(* CODESYS project 轮毂电机.project

Project tree, tasks and I/O mapping:
  Device : AM521-0808TP/TN, Shenzhen Inovance Control Technology, version 3.5.11.50
      settings: PersistentStartAdddr = 0; PersistentStartEndAddr = 524287; Mode = 0
    application Application
      libraries: Standard, * (System); IoDrvCANopenAxis, 1.11.4.0 (Inovance); HC_CANBus, 0.1.3.0 (Inovance); Util, 3.5.11.0 (System); SM3_Drive_ETC_Inovance, 1.0.5.0 (Inovance)
      task MainTask (cyclic, interval t#4ms, priority 1) calls main
      task CANOPEN (cyclic, interval t#10ms, priority 2) calls CANOpen_Task
      program main [ST]
      DifferentialMonitor
      program CANOpen_Task [ST]
      global variables GVL
      function block FB_AckermannKinematics [ST]
      trace Trace (task MainTask): Rr_Wheel.diActVelocity
      function block FB_CommandLimiter [ST]
      function block FB_SteerPositionPID [ST]
      function block FB_RearWheelVelocityPID [ST]
      function block FB_AckermannInverseKinematics [ST]
      function block FB_UDP [ST]
      function block FB_PWM [ST]
      function block FB_CAN_SCU_1 [ST]
      function block FB_Test [ST]
      function block FB_MoveByYaokong [ST]
      function block FB_MoveByFSD [ST]
      function block FB_CAN_CCU [ST]
      function block FB_UDP_Recv [ST]
      function block FB_UDP_Send [ST]
      function block test [ST]
      function block FB_CAN_VCU_SES_Req [ST]
      function block FB_CAN_BMS [ST]
      function block cantesttest [LD]
    ConfigStorage
    Resources List
    Device Diagnosis
    Network Configuration
      LocalBus Config
    HardWare Configuration
    SoftMotion General Axis Pool
    Local Bus
      GL20_2CAN : GL20 2通道CAN通信接口模块, Inovance, order no. 01440308, version 00.00.00.10
          settings: ModuleBaseInfoStruct.BusType = 10; ModuleBaseInfoStruct.RackNumber = 1; ModuleBaseInfoStruct.SlotNumber = 1; COMPort1 = 32; COMPort2 = 33; devGuid1 = 'e5bf4089-cd92-4763-8943-9d7dacf300b6'; devGuid2 = '326b6049-3dfc-42ac-adce-35d035554d5f'
          unmapped channels: RxPDO_CH, TxPDO_CH
    CAN : CAN总线, INOVANCE, version 00.00.00.10
      CAN_Port : CAN Port, Inovance, version 00.00.00.10
          settings: IsFreeCAN = False; DeviceGuid = '83de0e76-e450-4053-a235-86c09473ce3d'; DeviceName = 'GE20_CAN_485'; InterfaceNo = 1; Device = 'AM521-0808TP/TN'; Port = 4; Type = 41108
        CANopen主站 : CANopen主站, Inovance, version 00.00.00.10
            settings: COPManagerSyncStruct.SyncType = 1; COPManagerSyncStruct.SyncPeriod = 10000; COPManagerHeartbeatStruct.Enable = 1; Port NO = 4; IsPortSub = True; IsMainCAN = False; IsCANExt = True; IsLocalCAN = False
          C6049 : CANopen Slaver, Inovance, order no. 1525, version 00.00.00.10
              settings: NodeID = 3; EnableExpertSettings = 1; Error Control.SlaveHeartbeat.ProduceTime = 300; Error Control.SlaveHeartbeat.NrofConsumer = 1; VendorID = 1097; ProductNumber = 1; RevisionNumber = 131075; NrofRxPDO = 4; ValidRxPDO = 2; PdoCommuIndex = 5120; CanId = 515; TxType = 255;  = 1;  = 805306432; PdoCommuIndex = 5121; CanId = 771; TxType = 255;  = 1;  = 805371968; PdoCommuIndex = 5122; CanId = 1027; TxType = 255;  = 1;  = 805437504; PdoCommuIndex = 5123; CanId = 1283; TxType = 255;  = 1;  = 805503040; NrofTxPDO = 4; ValidTxPDO = 3; PdoCommuIndex = 6144; CanId = 387; TxType = 255; InhibitTime = 50;  = 1;  = 805568576; PdoCommuIndex = 6145; CanId = 643; TxType = 255;
                InhibitTime = 50;  = 1;  = 805634112; PdoCommuIndex = 6146; CanId = 899; TxType = 255; InhibitTime = 50;  = 1;  = 805699648; PdoCommuIndex = 6147; CanId = 1155; TxType = 255; InhibitTime = 50;  = 1;  = 805765184; SdoTimeout = 1000; NrofSDO = 31; SdoCommParam = 269877536; SdoErrHandle = 2; SdoJumptoLine = 31; SdoCommParam = 269942800; SdoCommValue = 300; SdoErrHandle = 2; SdoJumptoLine = 31; SdoCommParam = 269746208; SdoCommValue = 2147483779; SdoErrHandle = 2; SdoJumptoLine = 31; SdoCommParam = 269746208; SdoCommValue = 131; SdoErrHandle = 2; SdoJumptoLine = 31; SdoCommParam = 335544608; SdoCommValue = 2147484163; SdoErrHandle = 2; SdoJumptoLine = 31; SdoCommParam = 335610144; SdoCommValue = 2147484419; SdoErrHandle = 2; SdoJumptoLine = 31;
                SdoCommParam = 335610376; SdoCommValue = 255; SdoErrHandle = 2; SdoJumptoLine = 31; SdoCommParam = 369164296; SdoErrHandle = 2; SdoJumptoLine = 31; SdoCommParam = 369164576; SdoCommValue = 805371968; SdoErrHandle = 2; SdoJumptoLine = 31; SdoCommParam = 369164296; SdoCommValue = 1; SdoErrHandle = 2; SdoJumptoLine = 31; SdoCommParam = 335610144; SdoCommValue = 771; SdoErrHandle = 2; SdoJumptoLine = 31; SdoCommParam = 335675680; SdoCommValue = 2147484675; SdoErrHandle = 2; SdoJumptoLine = 31; SdoCommParam = 335741216; SdoCommValue = 2147484931; SdoErrHandle = 2; SdoJumptoLine = 31; SdoCommParam = 402653472; SdoCommValue = 2147484035; SdoErrHandle = 2; SdoJumptoLine = 31; SdoCommParam = 402653704; SdoCommValue = 255; SdoErrHandle = 2; SdoJumptoLine = 31; SdoCommParam = 402653968; SdoCommValue = 50; SdoErrHandle = 2; SdoJumptoLine = 31; SdoCommParam = 402654480;
                SdoErrHandle = 2; SdoJumptoLine = 31; SdoCommParam = 436207624; SdoErrHandle = 2; SdoJumptoLine = 31; SdoCommParam = 436207904; SdoCommValue = 805568576; SdoErrHandle = 2; SdoJumptoLine = 31; SdoCommParam = 436207624; SdoCommValue = 1; SdoErrHandle = 2; SdoJumptoLine = 31; SdoCommParam = 402653472; SdoCommValue = 387; SdoErrHandle = 2; SdoJumptoLine = 31; SdoCommParam = 402719008; SdoCommValue = 2147484291; SdoErrHandle = 2; SdoJumptoLine = 31; SdoCommParam = 402719240; SdoCommValue = 255; SdoErrHandle = 2; SdoJumptoLine = 31; SdoCommParam = 402719504; SdoCommValue = 50; SdoErrHandle = 2; SdoJumptoLine = 31; SdoCommParam = 402720016; SdoErrHandle = 2; SdoJumptoLine = 31; SdoCommParam = 436273160; SdoErrHandle = 2; SdoJumptoLine = 31; SdoCommParam = 436273440; SdoCommValue = 805634112; SdoErrHandle = 2; SdoJumptoLine = 31; SdoCommParam = 436273160;
                SdoCommValue = 1; SdoErrHandle = 2; SdoJumptoLine = 31; SdoCommParam = 402719008; SdoCommValue = 643; SdoErrHandle = 2; SdoJumptoLine = 31; SdoCommParam = 402784544; SdoCommValue = 2147484547; SdoErrHandle = 2; SdoJumptoLine = 31; SdoCommParam = 402850080; SdoCommValue = 2147484803; SdoErrHandle = 2; SdoJumptoLine = 31; FileName = 'C6049.eds'; FileVersion = '0x02'; FileRevision = '0x01'; EDSVersion = '4.0'; Description = 'EDS for 6049  Canopen Slave'; EDS File Path = 'D:\Asoftware\InoProShop\CODESYS\Common\AM600 Data\EdsFile\C6049.eds'; EDSVersion = 'EDLS'; VendorNumber = 1097; ProductName = 'C6049'; ProductNumber = 1; RevisionNumber = 131075; OrderCode = '60'; Baudrate = 368; SimpleBootUpSlave = 1; Granularity = 0; DynamicChannelsSupported = 0; GroupMessaging = 0; NrOfRXPDO = 4; NrOfTXPDO = 4; LSS_Supported = 0; DummyUsage = 0; SDOType = 0; SDOName = 'Set Heartbeat Consumer'; SDOType = 0; SDOName = 'Set Heartbeat Producer';
                SDOType = 0; SDOName = 'Disable Emcy COB-ID'; SDOType = 0; SDOName = 'Set Emcy COB-ID'; SDOType = 0; SDOName = 'Disable PDO'; SDOType = 0; SDOName = 'Disable PDO'; SDOType = 0; SDOName = 'Set transmission type'; SDOType = 0; SDOName = 'Clear PDO mapping'; SDOType = 0; SDOName = 'Set mapping'; SDOType = 0; SDOName = 'Set number of pdos'; SDOType = 0; SDOName = 'Set and enable COB-ID'; SDOType = 0; SDOName = 'Disable PDO'; SDOType = 0; SDOName = 'Disable PDO'; SDOType = 0; SDOName = 'Disable PDO'; SDOType = 0; SDOName = 'Set transmission type'; SDOType = 0; SDOName = 'Set inhibit time'; SDOType = 0; SDOName = 'Set event time'; SDOType = 0; SDOName = 'Clear PDO mapping'; SDOType = 0; SDOName = 'Set mapping'; SDOType = 0; SDOName = 'Set number of pdos'; SDOType = 0; SDOName = 'Set and enable COB-ID'; SDOType = 0; SDOName = 'Disable PDO';
                SDOType = 0; SDOName = 'Set transmission type'; SDOType = 0; SDOName = 'Set inhibit time'; SDOType = 0; SDOName = 'Set event time'; SDOType = 0; SDOName = 'Clear PDO mapping'; SDOType = 0; SDOName = 'Set mapping'; SDOType = 0; SDOName = 'Set number of pdos'; SDOType = 0; SDOName = 'Set and enable COB-ID'; SDOType = 0; SDOName = 'Disable PDO'; SDOType = 0; SDOName = 'Disable PDO'; Recv PDO Mapping Name.Recv PDO Mapping Name = '64 DI0'; Recv PDO Mapping Name.Recv PDO Mapping Name = '64 DI1'; Recv PDO Mapping Name.Recv PDO Mapping Name = '64 AI0'; Recv PDO Mapping Name.Recv PDO Mapping Name = '64 AI1'; Send PDO Mapping Name.Send PDO Mapping Name = '64 DO0'; Send PDO Mapping Name.Send PDO Mapping Name = '64 DO1'; Send PDO Mapping Name.Send PDO Mapping Name = '64 AO0'; Send PDO Mapping Name.Send PDO Mapping Name = '64 AO1'; Is Manual change COB-ID = 0; Is Manual change COB-ID = 0; Is Manual change COB-ID = 0; Is Manual change COB-ID = 0; Is Manual change COB-ID = 0; Is Manual change COB-ID = 0; Is Manual change COB-ID = 0; Is Manual change COB-ID = 0; MandatoryObjs = 3; Object Dictionary Item = '1000;Device Type;0x00000000;7;7;RO;0;-1;-1;-1'; Object Dictionary Item = '1001;Error Register;0x0;5;7;RO;0;-1;-1;-1'; Object Dictionary Item = '1018;Identity Object;;-1;9;;-1;4;-1;-1'; Object Dictionary Item = '1018sub0;number of entries;3;5;7;RO;0;-1;4;1'; Object Dictionary Item = '1018sub1;Vendor ID;0x00000449;7;7;RO;0;-1;-1;-1';
                Object Dictionary Item = '1018sub2;Product code;0x00000001;7;7;RO;0;-1;-1;-1'; Object Dictionary Item = '1018sub3;Revision number;0x00020003;7;7;RO;0;-1;-1;-1'; ManufacturerObjs = 9; Object Dictionary Item = '2000;Index 0x2000;;-1;9;;-1;2;-1;-1'; Object Dictionary Item = '2000sub0;Set TXPDO inhibit time;0x01;5;7;RO;0;-1;-1;-1'; Object Dictionary Item = '2000sub1;TXPDO1 inhibit time;100;5;7;RW;0;-1;-1;-1'; Object Dictionary Item = '3000;64 DI0;0;27;7;RO;1;-1;-1;-1'; Object Dictionary Item = '3001;64 DI1;0x0;27;7;RO;1;-1;-1;-1'; Object Dictionary Item = '3002;64 AI0;0;27;7;RO;1;-1;-1;-1'; Object Dictionary Item = '3003;64 AI1;0x0;27;7;RO;1;-1;-1;-1'; Object Dictionary Item = '3004;64 DO0;0x0;27;7;RWW;1;-1;-1;-1'; Object Dictionary Item = '3005;64 DO1;0x0;27;7;RWW;1;-1;-1;-1'; Object Dictionary Item = '3006;64 AO0;0x0;27;7;RWW;1;-1;-1;-1'; Object Dictionary Item = '3007;64 AO1;0x0;27;7;RWW;1;-1;-1;-1'; OptionsObjs = 20; Object Dictionary Item = '1005;COB-ID SYNC message;0x80;7;7;RW;0;-1;-1;-1'; Object Dictionary Item = '1008;Device Name;4055;9;7;CONST;0;-1;-1;-1'; Object Dictionary Item = '1016;Consumer Heartbeat time group;;-1;8;;-1;2;-1;-1'; Object Dictionary Item = '1016sub0;Number of entries;1;5;7;RO;0;-1;-1;-1'; Object Dictionary Item = '1016sub1;Consumer Heartbeat time;0;7;7;RW;0;-1;-1;-1'; Object Dictionary Item = '1017;Producer Heartbeat time group;0;6;7;RW;0;-1;-1;-1'; Object Dictionary Item = '1400;Receive PDO1 parameter;;-1;9;;-1;4;-1;-1'; Object Dictionary Item = '1400sub0;Number of entries;3;5;7;RO;0;-1;-1;-1'; Object Dictionary Item = '1400sub1;COB-ID;$NodeID + 0x200;7;7;RW;0;-1;-1;-1'; Object Dictionary Item = '1400sub2;Transmission type;255;5;7;RW;0;-1;-1;-1'; Object Dictionary Item = '1400sub3;Inhibit timer;0;5;7;RW;0;-1;-1;-1'; Object Dictionary Item = '1600;Receive PDO1 mapping;;-1;9;;-1;2;-1;-1'; Object Dictionary Item = '1600sub0;Number of mapped objects;0x1;5;7;RO;0;-1;5;0'; Object Dictionary Item = '1600sub1;1.mapped object;0x30000040;7;7;RO;0;-1;-1;-1'; Object Dictionary Item = '1401;Receive PDO2 parameter;;-1;9;;-1;4;-1;-1'; Object Dictionary Item = '1401sub0;Number of entries;3;5;7;RO;0;-1;-1;-1'; Object Dictionary Item = '1401sub1;COB-ID;$NodeID + 0x300;7;7;RW;0;-1;-1;-1'; Object Dictionary Item = '1401sub2;Transmission type;255;5;7;RW;0;-1;-1;-1'; Object Dictionary Item = '1401sub3;Inhibit timer;0;5;7;RW;0;-1;-1;-1'; Object Dictionary Item = '1601;Receive PDO2 mapping;;-1;9;;-1;2;-1;-1'; Object Dictionary Item = '1601sub0;Number of mapped objects;0x1;5;7;RO;0;-1;5;0'; Object Dictionary Item = '1601sub1;1.mapped object;0x30010040;7;7;RO;0;-1;-1;-1'; Object Dictionary Item = '1402;Receive PDO3 parameter;;-1;9;;-1;4;-1;-1'; Object Dictionary Item = '1402sub0;Number of entries;3;5;7;RO;0;-1;-1;-1'; Object Dictionary Item = '1402sub1;COB-ID;$NodeID + 0x400;7;7;RW;0;-1;-1;-1';
                Object Dictionary Item = '1402sub2;Transmission type;255;5;7;RW;0;-1;-1;-1'; Object Dictionary Item = '1402sub3;Inhibit timer;0;5;7;RW;0;-1;-1;-1'; Object Dictionary Item = '1602;Receive PDO3 mapping;;-1;9;;-1;2;-1;-1'; Object Dictionary Item = '1602sub0;Number of mapped objects;0x1;5;7;RO;0;-1;5;0'; Object Dictionary Item = '1602sub1;1.mapped object;0x30020040;7;7;RO;0;-1;-1;-1'; Object Dictionary Item = '1403;Receive PDO4 parameter;;-1;9;;-1;4;-1;-1'; Object Dictionary Item = '1403sub0;Number of entries;3;5;7;RO;0;-1;-1;-1'; Object Dictionary Item = '1403sub1;COB-ID;$NodeID + 0x500;7;7;RW;0;-1;-1;-1'; Object Dictionary Item = '1403sub2;Transmission type;255;5;7;RW;0;-1;-1;-1'; Object Dictionary Item = '1403sub3;Inhibit timer;0;5;7;RW;0;-1;-1;-1'; Object Dictionary Item = '1603;Receive PDO4 mapping;;-1;9;;-1;2;-1;-1'; Object Dictionary Item = '1603sub0;Number of mapped objects;0x1;5;7;RO;0;-1;5;0'; Object Dictionary Item = '1603sub1;1.mapped object;0x30030040;7;7;RO;0;-1;-1;-1'; Object Dictionary Item = '1800;Transmit PDO1 parameter;;-1;9;;-1;5;-1;-1'; Object Dictionary Item = '1800sub0;Number of entries;0x5;5;7;RO;0;-1;-1;-1'; Object Dictionary Item = '1800sub1;COB-ID;$NodeID + 0x180;7;7;RW;0;-1;-1;-1'; Object Dictionary Item = '1800sub2;Transmission type;255;5;7;RW;0;-1;-1;-1'; Object Dictionary Item = '1800sub3;Inhibit timer;50;6;7;RW;0;-1;-1;-1'; Object Dictionary Item = '1800sub5;Event Timer;0;27;7;RW;0;-1;65535;0'; Object Dictionary Item = '1A00;Transmit PDO1 mapping;;-1;9;;-1;2;-1;-1'; Object Dictionary Item = '1A00sub0;Number of mapped objects;0x1;5;7;RO;0;-1;4;0'; Object Dictionary Item = '1A00sub1;1.mapped object;0x30040040;7;7;RO;0;-1;-1;-1'; Object Dictionary Item = '1801;Transmit PDO2 parameter;;-1;9;;-1;5;-1;-1'; Object Dictionary Item = '1801sub0;Number of entries;0x5;5;7;RO;0;-1;-1;-1'; Object Dictionary Item = '1801sub1;COB-ID;$NodeID + 0x280;7;7;RW;0;-1;-1;-1'; Object Dictionary Item = '1801sub2;Transmission type;255;5;7;RW;0;-1;-1;-1'; Object Dictionary Item = '1801sub3;Inhibit timer;50;6;7;RW;0;-1;-1;-1'; Object Dictionary Item = '1801sub5;Event Timer;0;27;7;RW;0;-1;65535;0'; Object Dictionary Item = '1A01;Transmit PDO2 mapping;;-1;9;;-1;2;-1;-1'; Object Dictionary Item = '1A01sub0;Number of mapped objects;0x1;5;7;RO;0;-1;4;0'; Object Dictionary Item = '1A01sub1;1.mapped object;0x30050040;7;7;RO;0;-1;-1;-1'; Object Dictionary Item = '1802;Transmit PDO3 parameter;;-1;9;;-1;5;-1;-1'; Object Dictionary Item = '1802sub0;Number of entries;0x5;5;7;RO;0;-1;-1;-1'; Object Dictionary Item = '1802sub1;COB-ID;$NodeID + 0x380;7;7;RW;0;-1;-1;-1'; Object Dictionary Item = '1802sub2;Transmission type;255;5;7;RW;0;-1;-1;-1'; Object Dictionary Item = '1802sub3;Inhibit timer;50;6;7;RW;0;-1;-1;-1'; Object Dictionary Item = '1802sub5;Event Timer;0;27;7;RW;0;-1;65535;0'; Object Dictionary Item = '1A02;Transmit PDO3 mapping;;-1;9;;-1;2;-1;-1'; Object Dictionary Item = '1A02sub0;Number of mapped objects;0x1;5;7;RO;0;-1;4;0'; Object Dictionary Item = '1A02sub1;1.mapped object;0x30060040;7;7;RO;0;-1;-1;-1';
                Object Dictionary Item = '1803;Transmit PDO4 parameter;;-1;9;;-1;5;-1;-1'; Object Dictionary Item = '1803sub0;Number of entries;0x5;5;7;RO;0;-1;-1;-1'; Object Dictionary Item = '1803sub1;COB-ID;$NodeID + 0x480;7;7;RW;0;-1;-1;-1'; Object Dictionary Item = '1803sub2;Transmission type;255;5;7;RW;0;-1;-1;-1'; Object Dictionary Item = '1803sub3;Inhibit timer;50;6;7;RW;0;-1;-1;-1'; Object Dictionary Item = '1803sub5;Event Timer;0;27;7;RW;0;-1;65535;0'; Object Dictionary Item = '1A03;Transmit PDO4 mapping;;-1;9;;-1;2;-1;-1'; Object Dictionary Item = '1A03sub0;Number of mapped objects;0x1;5;7;RO;0;-1;4;0'; Object Dictionary Item = '1A03sub1;1.mapped object;0x30070040;7;7;RO;0;-1;-1;-1'
              output Application.YkqRxPDO0_data : LWORD  // 64 DI1
              input  Application.YkqTxPDO0_data : LWORD  // 64 DO0
              input  Application.Emergency_Stop : BOOL  // 64 DO0.Bit0
              input  Application.DriveByYaokong : BOOL  // 64 DO0.Bit10
              input  Application.DriveBySelf : BOOL  // 64 DO0.Bit11
              input  Application.Remote_Break : BOOL  // 64 DO0.Bit15
              input  Application.YkqTxPDO1_data : LWORD  // 64 DO1
          FDKServo_PMSM : CANopen Slaver, Inovance, order no. 1525, version 00.00.00.10
              settings: NodeID = 2; EnableExpertSettings = 1; Error Control.SlaveHeartbeat.ProduceTime = 300; Error Control.SlaveHeartbeat.NrofConsumer = 1; DeviceType = 131474; VendorID = 1459275; ProductNumber = 66128; NrofRxPDO = 4; ValidRxPDO = 3; PdoCommuIndex = 5120; CanId = 514; TxType = 255;  = 3;  = 1614807056;  = 1627324448;  = 1616904200; PdoCommuIndex = 5121; CanId = 770; TxType = 255;  = 2;  = 1618608160;  = 1619001376; PdoCommuIndex = 5122; CanId = 1026; TxType = 255;  = 0; PdoCommuIndex = 5123; CanId = 1282; TxType = 255;  = 0; NrofTxPDO = 4; ValidTxPDO = 3; PdoCommuIndex = 6144; CanId = 386; TxType = 255; InhibitTime = 100; EventTime = 10;  = 4;  = 1614872592;  = 536870928;
                 = 536936464;  = 1616969736; PdoCommuIndex = 6145; CanId = 642; TxType = 255; InhibitTime = 100; EventTime = 10;  = 2;  = 1617166368;  = 1617690656; PdoCommuIndex = 6146; CanId = 898; TxType = 255; InhibitTime = 100; EventTime = 10;  = 0; PdoCommuIndex = 6147; CanId = 1154; TxType = 255; InhibitTime = 100; EventTime = 10;  = 0; SdoTimeout = 1000; NrofSDO = 44; SdoCommParam = 268763168; SdoCommValue = 128; SdoCommParam = 269877536; SdoCommParam = 269942800; SdoCommValue = 300; SdoCommParam = 269746208; SdoCommValue = 2147483778; SdoCommParam = 269746208; SdoCommValue = 130; SdoCommParam = 335544608; SdoCommValue = 2147484162; SdoCommParam = 335544840; SdoCommValue = 255; SdoCommParam = 369098760; SdoCommParam = 369099040; SdoCommValue = 1614807056;
                SdoCommParam = 369099296; SdoCommValue = 1627324448; SdoCommParam = 369099552; SdoCommValue = 1616904200; SdoCommParam = 369098760; SdoCommValue = 3; SdoCommParam = 335544608; SdoCommValue = 514; SdoCommParam = 335610144; SdoCommValue = 2147484418; SdoCommParam = 335610376; SdoCommValue = 255; SdoCommParam = 369164296; SdoCommParam = 369164576; SdoCommValue = 1618608160; SdoCommParam = 369164832; SdoCommValue = 1619001376; SdoCommParam = 369164296; SdoCommValue = 2; SdoCommParam = 335610144; SdoCommValue = 770; SdoCommParam = 335675680; SdoCommValue = 2147484674; SdoCommParam = 335741216; SdoCommValue = 2147484930; SdoCommParam = 402653472; SdoCommValue = 2147484034; SdoCommParam = 402653704; SdoCommValue = 255; SdoCommParam = 402653968; SdoCommValue = 100; SdoCommParam = 402654480; SdoCommValue = 10; SdoCommParam = 436207624; SdoCommParam = 436207904; SdoCommValue = 1614872592; SdoCommParam = 436208160; SdoCommValue = 536870928; SdoCommParam = 436208416; SdoCommValue = 536936464;
                SdoCommParam = 436208672; SdoCommValue = 1616969736; SdoCommParam = 436207624; SdoCommValue = 4; SdoCommParam = 402653472; SdoCommValue = 386; SdoCommParam = 402719008; SdoCommValue = 2147484290; SdoCommParam = 402719240; SdoCommValue = 255; SdoCommParam = 402719504; SdoCommValue = 100; SdoCommParam = 402720016; SdoCommValue = 10; SdoCommParam = 436273160; SdoCommParam = 436273440; SdoCommValue = 1617166368; SdoCommParam = 436273696; SdoCommValue = 1617690656; SdoCommParam = 436273160; SdoCommValue = 2; SdoCommParam = 402719008; SdoCommValue = 642; SdoCommParam = 402784544; SdoCommValue = 2147484546; SdoCommParam = 402850080; SdoCommValue = 2147484802; FileName = 'FDK_PMSM.eds'; FileVersion = '0x01'; FileRevision = '0x01'; EDSVersion = '4.0'; Description = 'EDS for FDK_Single_DRIVER'; EDS File Path = 'D:\Asoftware\InoProShop\CODESYS\Common\AM600 Data\EdsFile\FDK_PMSM_SIEMENS-VSXXDXX-A-20240203.eds'; EDSVersion = 'FDK, INC.'; VendorNumber = 1459275; ProductName = 'FDKServo-PMSM'; ProductNumber = 66128; RevisionNumber = 0; OrderCode = 'DVPCOPM-SL'; Baudrate = 503;
                SimpleBootUpSlave = 1; Granularity = 8; DynamicChannelsSupported = 0; GroupMessaging = 0; NrOfRXPDO = 4; NrOfTXPDO = 4; LSS_Supported = 1; DummyUsage = 0; SDOType = 0; SDOName = 'Disable COB-ID sync'; SDOType = 0; SDOName = 'Set Heartbeat Consumer'; SDOType = 0; SDOName = 'Set Heartbeat Producer'; SDOType = 0; SDOName = 'Disable Emcy COB-ID'; SDOType = 0; SDOName = 'Set Emcy COB-ID'; SDOType = 0; SDOName = 'Disable PDO'; SDOType = 0; SDOName = 'Set transmission type'; SDOType = 0; SDOName = 'Clear PDO mapping'; SDOType = 0; SDOName = 'Set mapping'; SDOType = 0; SDOName = 'Set mapping'; SDOType = 0; SDOName = 'Set mapping'; SDOType = 0; SDOName = 'Set number of pdos'; SDOType = 0; SDOName = 'Set and enable COB-ID'; SDOType = 0; SDOName = 'Disable PDO'; SDOType = 0; SDOName = 'Set transmission type'; SDOType = 0; SDOName = 'Clear PDO mapping';
                SDOType = 0; SDOName = 'Set mapping'; SDOType = 0; SDOName = 'Set mapping'; SDOType = 0; SDOName = 'Set number of pdos'; SDOType = 0; SDOName = 'Set and enable COB-ID'; SDOType = 0; SDOName = 'Disable PDO'; SDOType = 0; SDOName = 'Disable PDO'; SDOType = 0; SDOName = 'Disable PDO'; SDOType = 0; SDOName = 'Set transmission type'; SDOType = 0; SDOName = 'Set inhibit time'; SDOType = 0; SDOName = 'Set event time'; SDOType = 0; SDOName = 'Clear PDO mapping'; SDOType = 0; SDOName = 'Set mapping'; SDOType = 0; SDOName = 'Set mapping'; SDOType = 0; SDOName = 'Set mapping'; SDOType = 0; SDOName = 'Set mapping'; SDOType = 0; SDOName = 'Set number of pdos'; SDOType = 0; SDOName = 'Set and enable COB-ID'; SDOType = 0; SDOName = 'Disable PDO'; SDOType = 0; SDOName = 'Set transmission type'; SDOType = 0; SDOName = 'Set inhibit time';
                SDOType = 0; SDOName = 'Set event time'; SDOType = 0; SDOName = 'Clear PDO mapping'; SDOType = 0; SDOName = 'Set mapping'; SDOType = 0; SDOName = 'Set mapping'; SDOType = 0; SDOName = 'Set number of pdos'; SDOType = 0; SDOName = 'Set and enable COB-ID'; SDOType = 0; SDOName = 'Disable PDO'; SDOType = 0; SDOName = 'Disable PDO'; Recv PDO Mapping Name.Recv PDO Mapping Name = 'Controlword'; Recv PDO Mapping Name.Recv PDO Mapping Name = 'Target Velocity'; Recv PDO Mapping Name.Recv PDO Mapping Name = 'Modes of operation'; Recv PDO Mapping Name.Recv PDO Mapping Name = 'Target Position'; Recv PDO Mapping Name.Recv PDO Mapping Name = 'Max motor speed'; Send PDO Mapping Name.Send PDO Mapping Name = 'Statusword'; Send PDO Mapping Name.Send PDO Mapping Name = 'FaultCode1'; Send PDO Mapping Name.Send PDO Mapping Name = 'WorkState1'; Send PDO Mapping Name.Send PDO Mapping Name = 'Modes Of Operation Display'; Send PDO Mapping Name.Send PDO Mapping Name = 'Position Actual Value'; Send PDO Mapping Name.Send PDO Mapping Name = 'Velocity actual value'; Is Manual change COB-ID = 0; Is Manual change COB-ID = 0; Is Manual change COB-ID = 0; Is Manual change COB-ID = 0; Is Manual change COB-ID = 0; Is Manual change COB-ID = 0; Is Manual change COB-ID = 0; Is Manual change COB-ID = 0; MandatoryObjs = 3; Object Dictionary Item = '1000;CAN Controller Type;0x20192;7;7;RO;0;-1;-1;-1'; Object Dictionary Item = '1001;Error Register;0;5;7;RO;0;-1;-1;-1'; Object Dictionary Item = '1018;Identity Object;;-1;9;;-1;4;-1;-1'; Object Dictionary Item = '1018sub0;number of entries;3;5;7;RO;0;-1;4;1';
                Object Dictionary Item = '1018sub1;Vendor ID;0x0016444B;7;7;RO;0;-1;-1;-1'; Object Dictionary Item = '1018sub2;Product code;0x00010250;7;7;RO;0;-1;-1;-1'; Object Dictionary Item = '1018sub3;Revision number;0x00000000;7;7;RO;0;-1;-1;-1'; ManufacturerObjs = 30; Object Dictionary Item = '2000;FaultCode1;;6;7;RO;1;-1;65535;0'; Object Dictionary Item = '2001;WorkState1;;6;7;RO;1;-1;65535;0'; Object Dictionary Item = '2002;Motor_T;;6;7;RO;1;-1;-1;-1'; Object Dictionary Item = '2004;WARN;;6;7;RO;1;-1;65535;0'; Object Dictionary Item = '2005;CurrentBase;;6;7;RO;1;-1;65535;0'; Object Dictionary Item = '2006;LineEncoder;;4;7;RO;1;-1;65535;0'; Object Dictionary Item = '2007;Feedback Type;;6;7;RW;0;-1;65535;0'; Object Dictionary Item = '2008;Pole Pairs;;6;7;RW;0;-1;65535;0'; Object Dictionary Item = '2009;CAN ID;;5;7;RW;0;-1;-1;-1'; Object Dictionary Item = '200A;Can Baud Rate;;6;7;RW;0;-1;-1;-1'; Object Dictionary Item = '200B;Rated Current;;3;7;RW;0;-1;-1;-1'; Object Dictionary Item = '200C;Rated Speed;;3;7;RW;0;-1;-1;-1'; Object Dictionary Item = '200D;Overload Current;;6;7;RW;1;-1;-1;-1'; Object Dictionary Item = '200E;Overload Time;;6;7;RW;1;-1;-1;-1'; Object Dictionary Item = '200F;Current Loop P;;6;7;RW;1;-1;-1;-1'; Object Dictionary Item = '2010;Current Loop I;;6;7;RW;1;-1;-1;-1'; Object Dictionary Item = '2011;Speed Loop p0;;6;7;RW;1;-1;-1;-1'; Object Dictionary Item = '2012;Speed Loop P1;;6;7;RW;1;-1;-1;-1'; Object Dictionary Item = '2013;Speed Loop I;;6;7;RW;1;-1;-1;-1'; Object Dictionary Item = '2014;Position Loop P0;;6;7;RW;1;-1;-1;-1'; Object Dictionary Item = '2015;Position Loop P1;;6;7;RW;1;-1;-1;-1'; Object Dictionary Item = '2016;Command0;;6;7;RW;1;-1;-1;-1'; Object Dictionary Item = '2017;Command1;;6;7;RW;1;-1;-1;-1'; Object Dictionary Item = '2018;Software Limited Cache;;6;7;RW;1;-1;-1;-1'; Object Dictionary Item = '2019;Software Limited Forward Position;;4;7;RW;1;-1;-1;-1'; Object Dictionary Item = '201A;Software Limited Reverse Position;;4;7;RW;1;-1;-1;-1'; Object Dictionary Item = '201B;RS485_NodeID;;6;7;RW;1;-1;-1;-1'; Object Dictionary Item = '201C;RS485_Baudrate;;6;7;RW;1;-1;-1;-1'; Object Dictionary Item = '201D;RS485_Protocol;;6;7;RW;1;-1;-1;-1'; Object Dictionary Item = '22A2;System_T;;6;7;RO;1;-1;-1;-1'; OptionsObjs = 104; Object Dictionary Item = '1002;Manufacturer Status Register;;7;7;RO;1;-1;-1;-1'; Object Dictionary Item = '1003;Pre-defined Error Field;;-1;8;;-1;17;-1;-1'; Object Dictionary Item = '1003sub0;Number of Errors;0;5;7;RW;0;-1;16;0'; Object Dictionary Item = '1003sub1;Standard Error Field;0;7;7;RO;0;-1;-1;0'; Object Dictionary Item = '1003sub2;Standard Error Field;0;7;7;RO;0;-1;-1;0';
                Object Dictionary Item = '1003sub3;Standard Error Field;0;7;7;RO;0;-1;-1;0'; Object Dictionary Item = '1003sub4;Standard Error Field;0;7;7;RO;0;-1;-1;0'; Object Dictionary Item = '1003sub5;Standard Error Field;0;7;7;RO;0;-1;-1;0'; Object Dictionary Item = '1003sub6;Standard Error Field;0;7;7;RO;0;-1;-1;0'; Object Dictionary Item = '1003sub7;Standard Error Field;0;7;7;RO;0;-1;-1;0'; Object Dictionary Item = '1003sub8;Standard Error Field;0;7;7;RO;0;-1;-1;0'; Object Dictionary Item = '1003sub9;Standard Error Field;0;7;7;RO;0;-1;-1;0'; Object Dictionary Item = '1003suba;Standard Error Field;0;7;7;RO;0;-1;-1;0'; Object Dictionary Item = '1003subb;Standard Error Field;0;7;7;RO;0;-1;-1;0'; Object Dictionary Item = '1003subc;Standard Error Field;0;7;7;RO;0;-1;-1;0'; Object Dictionary Item = '1003subd;Standard Error Field;0;7;7;RO;0;-1;-1;0'; Object Dictionary Item = '1003sube;Standard Error Field;0;7;7;RO;0;-1;-1;0'; Object Dictionary Item = '1003subf;Standard Error Field;0;7;7;RO;0;-1;-1;0'; Object Dictionary Item = '1003sub10;Standard Error Field;0;7;7;RO;0;-1;-1;0'; Object Dictionary Item = '1005;COB-ID SYNC-message;0x80;7;7;RW;0;-1;-1;-1'; Object Dictionary Item = '1006;Communication Cycle Period;0;7;7;RW;0;-1;-1;0'; Object Dictionary Item = '1008;Manufacturer Device Name;;9;7;CONST;0;-1;-1;-1'; Object Dictionary Item = '1009;Manufacturer Hardware Version;;9;7;CONST;0;-1;-1;-1'; Object Dictionary Item = '100A;Manufacturer Software Version;;9;7;CONST;0;-1;-1;-1'; Object Dictionary Item = '100B;Node-ID;1;5;7;RO;0;-1;127;1'; Object Dictionary Item = '1010;Store Parameters;;-1;8;;-1;4;-1;-1'; Object Dictionary Item = '1010sub0;Largest Supported Sub-index;3;5;7;RO;0;-1;3;3'; Object Dictionary Item = '1010sub1;Save All Parameters;;7;7;RW;0;-1;-1;-1'; Object Dictionary Item = '1010sub2;Save Communication Parameters;0;7;7;RW;0;-1;-1;-1'; Object Dictionary Item = '1010sub3;Save ApplicationParameters;0;7;7;RW;0;-1;-1;-1'; Object Dictionary Item = '1011;Restore  Parameters;;-1;8;;-1;4;-1;-1'; Object Dictionary Item = '1011sub0;Largest Supported Sub-index;3;5;7;RO;0;-1;3;3'; Object Dictionary Item = '1011sub1;Restore All Parameters;;7;7;RW;0;-1;-1;-1'; Object Dictionary Item = '1011sub2;Restore Communication Parameters;0;7;7;RW;0;-1;-1;-1'; Object Dictionary Item = '1011sub3;Restore ApplicationParameters;0;7;7;RW;0;-1;-1;-1'; Object Dictionary Item = '1012;COB-ID Time Stamp Message;0x80000100;7;7;RW;0;-1;-1;-1'; Object Dictionary Item = '1013;High Resolution TimeStamp;0;7;7;RW;0;-1;-1;0'; Object Dictionary Item = '1014;COB-ID Emergency Message;$NODEID+0x80;7;7;RW;0;-1;-1;-1'; Object Dictionary Item = '1016;Consumer Heartbeat Time;;-1;8;;-1;2;-1;-1'; Object Dictionary Item = '1016sub0;Number of Entries;1;5;7;RO;0;-1;1;1'; Object Dictionary Item = '1016sub1;Consumer Heartbeat Time;0;7;7;RW;0;-1;-1;-1'; Object Dictionary Item = '1017;Producer heartbeat time;0;6;7;RW;0;-1;-1;-1'; Object Dictionary Item = '1023;OS Command;;-1;9;;-1;4;-1;-1'; Object Dictionary Item = '1023sub0;Number of Entries;3;5;7;RO;0;-1;3;3'; Object Dictionary Item = '1023sub1;Command;;10;7;WO;0;-1;-1;-1';
                Object Dictionary Item = '1023sub2;Status;0;5;7;RO;0;-1;255;0'; Object Dictionary Item = '1023sub3;Reply;;10;7;RO;0;-1;-1;-1'; Object Dictionary Item = '1024;OS Command Mode;0;5;7;WO;0;-1;-1;-1'; Object Dictionary Item = '1029;Error Behavior;;-1;8;;-1;2;-1;-1'; Object Dictionary Item = '1029sub0;Number of Error Classes;1;5;7;RO;0;-1;1;1'; Object Dictionary Item = '1029sub1;Communication Error;1;5;7;RW;0;-1;2;0'; Object Dictionary Item = '1200;1st Server SDO Parameter;;-1;9;;-1;3;-1;-1'; Object Dictionary Item = '1200sub0;Number of Entries;2;5;7;RO;0;-1;2;2'; Object Dictionary Item = '1200sub1;COB-ID Client->Server (Rx);$NODEID+0x600;7;7;RO;0;-1;-1;-1'; Object Dictionary Item = '1200sub2;COB-ID Server ->Client (Tx);$NODEID+0x580;7;7;RO;0;-1;-1;-1'; Object Dictionary Item = '1400;1st Receive PDO Parameter;;-1;9;;-1;3;-1;-1'; Object Dictionary Item = '1400sub0;Largest Sub-Index Supported;2;5;7;RO;0;-1;2;2'; Object Dictionary Item = '1400sub1;COB-ID Used by PDO;$NODEID+0x200;7;7;RW;0;-1;-1;-1'; Object Dictionary Item = '1400sub2;Transmission Type;0xFF;5;7;RW;0;-1;255;0'; Object Dictionary Item = '1600;1st Receive PDO Mapping;;-1;9;;-1;5;-1;-1'; Object Dictionary Item = '1600sub0;Number of Mapped Application Objects in PDO;3;5;7;RW;0;-1;8;0'; Object Dictionary Item = '1600sub1;PDO Mapping for the 1st Application Object to Be Mapped;0x60400010;7;7;RW;0;-1;-1;-1'; Object Dictionary Item = '1600sub2;PDO Mapping for the 2nd Application Object to Be Mapped;0x60FF0020;7;7;RW;0;-1;-1;-1'; Object Dictionary Item = '1600sub3;PDO Mapping for the 3rd Application Object to Be Mapped;0x60600008;7;7;RW;0;-1;-1;-1'; Object Dictionary Item = '1600sub4;PDO Mapping for the 4th Application Object to Be Mapped;;7;7;RW;0;-1;-1;-1'; Object Dictionary Item = '1401;2nd Receive PDO parameter;;-1;9;;-1;3;-1;-1'; Object Dictionary Item = '1401sub0;Number of Entries;2;5;7;RO;0;-1;2;2'; Object Dictionary Item = '1401sub1;COB-ID used by PDO;$NODEID+0x300;7;7;RW;0;-1;-1;-1'; Object Dictionary Item = '1401sub2;Transmission Type;0xFF;5;7;RW;0;-1;255;0'; Object Dictionary Item = '1601;2nd Receive PDO Mapping;;-1;9;;-1;5;-1;-1'; Object Dictionary Item = '1601sub0;Number of Mapped Application Objects in PDO;2;5;7;RW;0;-1;8;0'; Object Dictionary Item = '1601sub1;PDO Mapping for the 1st Application Object to Be Mapped;0x607A0020;7;7;RW;0;-1;-1;-1'; Object Dictionary Item = '1601sub2;PDO Mapping for the 2nd Application Object to Be Mapped;0x60800020;7;7;RW;0;-1;-1;-1'; Object Dictionary Item = '1601sub3;PDO Mapping for the 3rd Application Object to Be Mapped;;7;7;RW;0;-1;-1;-1'; Object Dictionary Item = '1601sub4;PDO Mapping for the 4th Application Object to Be Mapped;;7;7;RW;0;-1;-1;-1'; Object Dictionary Item = '1402;3rd Receive PDO Parameters;;-1;9;;-1;3;-1;-1'; Object Dictionary Item = '1402sub0;number of elements;2;5;7;RO;0;-1;2;2'; Object Dictionary Item = '1402sub1;COB-ID used by PDO;$NODEID+0x400;7;7;RW;0;-1;-1;-1'; Object Dictionary Item = '1402sub2;Transmission Type;0xFF;5;7;RW;0;-1;255;0'; Object Dictionary Item = '1602;3rd Receive PDO Mapping;;-1;9;;-1;5;-1;-1'; Object Dictionary Item = '1602sub0;Number of Mapped Application Objects in PDO;0;5;7;RW;0;-1;8;0'; Object Dictionary Item = '1602sub1;PDO Mapping for the 1st Application Object to Be Mapped;;7;7;RW;0;-1;-1;-1'; Object Dictionary Item = '1602sub2;PDO Mapping for the 2nd Application Object to Be Mapped;;7;7;RW;0;-1;-1;-1'; Object Dictionary Item = '1602sub3;PDO Mapping for the 3rd Application Object to Be Mapped;;7;7;RW;0;-1;-1;-1'; Object Dictionary Item = '1602sub4;PDO Mapping for the 4th Application Object to Be Mapped;;7;7;RW;0;-1;-1;-1';
                Object Dictionary Item = '1403;4th Received PDO Parameters;;-1;9;;-1;3;-1;-1'; Object Dictionary Item = '1403sub0;number of elements;2;5;7;RO;0;-1;2;2'; Object Dictionary Item = '1403sub1;COB-ID used by PDO;$NODEID+0x500;7;7;RW;0;-1;-1;-1'; Object Dictionary Item = '1403sub2;Transmission Type;0xFF;5;7;RW;0;-1;255;0'; Object Dictionary Item = '1603;4th Receive PDO Mapping;;-1;9;;-1;5;-1;-1'; Object Dictionary Item = '1603sub0;Number of Mapped Application Objects in PDO;0;5;7;RW;0;-1;8;0'; Object Dictionary Item = '1603sub1;PDO Mapping for the 1st Application Object to Be Mapped;;7;7;RW;0;-1;-1;-1'; Object Dictionary Item = '1603sub2;PDO Mapping for the 2nd Application Object to Be Mapped;;7;7;RW;0;-1;-1;-1'; Object Dictionary Item = '1603sub3;PDO Mapping for the 3rd Application Object to Be Mapped;;7;7;RW;0;-1;-1;-1'; Object Dictionary Item = '1603sub4;PDO Mapping for the 4th Application Object to Be Mapped;;7;7;RW;0;-1;-1;-1'; Object Dictionary Item = '1800;1st Transmit PDO Parameter;;-1;9;;-1;6;-1;-1'; Object Dictionary Item = '1800sub0;Largest Sub-Index Supported;5;5;7;RO;0;-1;5;5'; Object Dictionary Item = '1800sub1;COB-ID Used by PDO;$NODEID+0x00000180;7;7;RW;0;-1;-1;-1'; Object Dictionary Item = '1800sub2;Transmission Type;255;5;7;RW;0;-1;255;0'; Object Dictionary Item = '1800sub3;Inhibit Time;100;6;7;RW;0;-1;-1;-1'; Object Dictionary Item = '1800sub4;Reserved;;5;7;RW;0;-1;-1;-1'; Object Dictionary Item = '1800sub5;Event Timer;10;6;7;RW;0;-1;-1;-1'; Object Dictionary Item = '1A00;1st Transmit PDO Mapping;;-1;9;;-1;5;-1;-1'; Object Dictionary Item = '1A00sub0;Number Of Mapped Application Object In PDO.;4;5;7;RW;0;-1;8;0'; Object Dictionary Item = '1A00sub1;PDO Mapping For The 1st Application Object To Be Mapped;0x60410010;7;7;RW;0;-1;-1;-1'; Object Dictionary Item = '1A00sub2;PDO Mapping For The 2nd  Application Object To Be Mapped;0x20000010;7;7;RW;0;-1;-1;-1'; Object Dictionary Item = '1A00sub3;PDO Mapping For The 3rd Application Object To Be Mapped;0x20010010;7;7;RW;0;-1;-1;-1'; Object Dictionary Item = '1A00sub4;PDO Mapping For The 4th Application Object To Be Mapped;0x60610008;7;7;RW;0;-1;-1;-1'; Object Dictionary Item = '1801;2nd Transmit PDO Parameter;;-1;9;;-1;6;-1;-1'; Object Dictionary Item = '1801sub0;Largest Sub-Index Supported;5;5;7;RO;0;-1;5;5'; Object Dictionary Item = '1801sub1;COB-ID Used  by PDO;$NODEID+0x00000280;7;7;RW;0;-1;-1;-1'; Object Dictionary Item = '1801sub2;Transmission Type;255;5;7;RW;0;-1;255;0'; Object Dictionary Item = '1801sub3;Inhibit Time;100;6;7;RW;0;-1;-1;-1'; Object Dictionary Item = '1801sub4;Reserved;;5;7;RW;0;-1;-1;-1'; Object Dictionary Item = '1801sub5;Event Timer;10;6;7;RW;0;-1;-1;-1'; Object Dictionary Item = '1A01;2nd Transmit PDO Mapping;;-1;9;;-1;5;-1;-1'; Object Dictionary Item = '1A01sub0;Number Of Mapped Application Object In PDO.;2;5;7;RW;0;-1;8;0'; Object Dictionary Item = '1A01sub1;PDO Mapping For The 1st Application Object To Be Mapped;0x60640020;7;7;RW;0;-1;-1;-1'; Object Dictionary Item = '1A01sub2;PDO Mapping For The 2nd  Application Object To Be Mapped;0x606C0020;7;7;RW;0;-1;-1;-1'; Object Dictionary Item = '1A01sub3;PDO Mapping For The 3rd Application Object To Be Mapped;;7;7;RW;0;-1;-1;-1'; Object Dictionary Item = '1A01sub4;PDO Mapping For The 4th Application Object To Be Mapped;;7;7;RW;0;-1;-1;-1'; Object Dictionary Item = '1802;3rd Transmit PDO Parameter;;-1;9;;-1;6;-1;-1'; Object Dictionary Item = '1802sub0;Largest Sub-Index Supported;5;5;7;RO;0;-1;5;5'; Object Dictionary Item = '1802sub1;COB-ID Used  by PDO;$NODEID+0x00000380;7;7;RW;0;-1;-1;-1'; Object Dictionary Item = '1802sub2;Transmission Type;255;5;7;RW;0;-1;255;0';
                Object Dictionary Item = '1802sub3;Inhibit Time;100;6;7;RW;0;-1;-1;-1'; Object Dictionary Item = '1802sub4;Reserved;;5;7;RW;0;-1;-1;-1'; Object Dictionary Item = '1802sub5;Event Timer;10;6;7;RW;0;-1;-1;-1'; Object Dictionary Item = '1A02;3rd Transmit PDO  Mapping;;-1;9;;-1;5;-1;-1'; Object Dictionary Item = '1A02sub0;Number Of Mapped Application Object In PDO.;0;5;7;RW;0;-1;8;0'; Object Dictionary Item = '1A02sub1;PDO Mapping For The 1st Application Object To Be Mapped;;7;7;RW;0;-1;-1;-1'; Object Dictionary Item = '1A02sub2;PDO Mapping For The 2nd Application Object To Be Mapped;;7;7;RW;0;-1;-1;-1'; Object Dictionary Item = '1A02sub3;PDO Mapping For The 3rd Application Object To Be Mapped;;7;7;RW;0;-1;-1;-1'; Object Dictionary Item = '1A02sub4;PDO Mapping For The 4th Application Object To Be Mapped;;7;7;RW;0;-1;-1;-1'; Object Dictionary Item = '1803;4th Transmit PDO Parameter;;-1;9;;-1;6;-1;-1'; Object Dictionary Item = '1803sub0;Largest Sub-Index Supported;5;5;7;RO;0;-1;5;5'; Object Dictionary Item = '1803sub1;COB-ID Used  by PDO;$NODEID+0x00000480;7;7;RW;0;-1;-1;-1'; Object Dictionary Item = '1803sub2;Transmission Type;255;5;7;RW;0;-1;255;0'; Object Dictionary Item = '1803sub3;Inhibit Time;100;6;7;RW;0;-1;-1;-1'; Object Dictionary Item = '1803sub4;Reserved;;5;7;RW;0;-1;-1;-1'; Object Dictionary Item = '1803sub5;Event Timer;10;6;7;RW;0;-1;-1;-1'; Object Dictionary Item = '1A03;4th Transmit PDO  Mapping;;-1;9;;-1;5;-1;-1'; Object Dictionary Item = '1A03sub0;Number Of Mapped Application Object In PDO.;0;5;7;RW;0;-1;8;0'; Object Dictionary Item = '1A03sub1;PDO Mapping For The 1st Application Object To Be Mapped;;7;7;RW;0;-1;-1;-1'; Object Dictionary Item = '1A03sub2;PDO Mapping For The 2nd Application Object To Be Mapped;;7;7;RW;0;-1;-1;-1'; Object Dictionary Item = '1A03sub3;PDO Mapping For The 3rd Application Object To Be Mapped;;7;7;RW;0;-1;-1;-1'; Object Dictionary Item = '1A03sub4;PDO Mapping For The 4th Application Object To Be Mapped;;7;7;RW;0;-1;-1;-1'; Object Dictionary Item = '6007;Abort Connection Option Code;0;3;7;RW;0;-1;32767;-32768'; Object Dictionary Item = '603F;Error code;0;6;7;RO;0;-1;65535;0'; Object Dictionary Item = '6040;Controlword;;6;7;RWW;1;-1;65535;0'; Object Dictionary Item = '6041;Statusword;;6;7;RO;1;-1;65535;0'; Object Dictionary Item = '605A;Quick Stop Option Code;2;3;7;RW;0;-1;6;0'; Object Dictionary Item = '605B;Shutdown Option Code;0;3;7;RW;0;-1;1;0'; Object Dictionary Item = '605C;Disable Operation Option Code;1;3;7;RW;0;-1;1;0'; Object Dictionary Item = '605D;Halt Option Code;1;3;7;RW;0;-1;2;0'; Object Dictionary Item = '605E;Fault Reaction Option Code;0;3;7;RW;0;-1;0;0'; Object Dictionary Item = '6060;Modes of operation;;2;7;RWW;1;-1;7;-1'; Object Dictionary Item = '6061;Modes Of Operation Display;;2;7;RO;1;-1;7;-1'; Object Dictionary Item = '6062;Position Demand Value;0;4;7;RO;1;-1;2147483647;-1'; Object Dictionary Item = '6063;Position Actual Value;;4;7;RO;1;-1;2147483647;-1'; Object Dictionary Item = '6064;Position Actual Value;0;4;7;RO;1;-1;2147483647;-1'; Object Dictionary Item = '6065;Following Error Window;;7;7;RW;0;-1;-1;0'; Object Dictionary Item = '6066;Following Error Time Out;;6;7;RW;0;-1;65535;0'; Object Dictionary Item = '6067;Position Window;;7;7;RW;0;-1;32000;0'; Object Dictionary Item = '6068;Position Windows Time;;6;7;RW;0;-1;100;0';
                Object Dictionary Item = '6069;Velocity Sensor Actual Value;;4;7;RO;1;-1;-1;-1'; Object Dictionary Item = '606A;Sensor selection code;;3;7;RW;0;-1;1;0'; Object Dictionary Item = '606B;Velocity Demand Value;;4;7;RO;1;-1;-1;-1'; Object Dictionary Item = '606C;Velocity actual value;;4;7;RO;1;-1;-1;-1'; Object Dictionary Item = '606D;Velocity Window;;6;7;RW;0;-1;65535;0'; Object Dictionary Item = '606E;Velocity Window Time;;6;7;RW;0;-1;65535;0'; Object Dictionary Item = '606F;Velocity Threshold;;6;7;RW;0;-1;65535;0'; Object Dictionary Item = '6070;Velocity Threshold Time;;6;7;RW;0;-1;65535;0'; Object Dictionary Item = '6071;Target Torque;0;3;7;RWW;1;-1;-1;-1'; Object Dictionary Item = '6072;Max Torque;0;6;7;RW;0;-1;-1;-1'; Object Dictionary Item = '6073;Max Current;0;6;7;RW;0;-1;-1;-1'; Object Dictionary Item = '6074;Torque demand value;0;3;7;RO;1;-1;-1;-1'; Object Dictionary Item = '6075;Motor rated current;0;7;7;RW;0;-1;-1;-1'; Object Dictionary Item = '6076;Motor rated torque;0;7;7;RW;0;-1;-1;-1'; Object Dictionary Item = '6077;Torque actual value;0;3;7;RO;1;-1;-1;-1'; Object Dictionary Item = '6078;Current Actual Value;0;3;7;RO;1;-1;-1;-1'; Object Dictionary Item = '607A;Target Position;;4;7;RWW;1;-1;2147483647;-2147483648'; Object Dictionary Item = '607B;Position Range Limit;;-1;8;;-1;3;-1;-1'; Object Dictionary Item = '607Bsub0;Number of Entries;2;5;7;RO;0;-1;2;2'; Object Dictionary Item = '607Bsub1;Min Position Range Limit;-1000000000;4;7;RW;0;-1;-1;-1'; Object Dictionary Item = '607Bsub2;Max Position Range Limit;1000000000;4;7;RW;0;-1;-1;-1'; Object Dictionary Item = '607C;Home offset;0;4;7;RW;0;-1;2147483647;-2147483648'; Object Dictionary Item = '607D;Software Position Limit;;-1;8;;-1;3;-1;-1'; Object Dictionary Item = '607Dsub0;Number of Entries;2;5;7;RO;0;-1;2;2'; Object Dictionary Item = '607Dsub1;Min Position Limit;-1000000000;4;7;RW;0;-1;-1;-1'; Object Dictionary Item = '607Dsub2;Max Position Limit;1000000000;4;7;RW;0;-1;-1;-1'; Object Dictionary Item = '607E;Polarity;0;5;7;RWW;1;-1;-1;-1'; Object Dictionary Item = '607F;Max Profile Velocity;;7;7;RW;0;-1;-1;0'; Object Dictionary Item = '6080;Max motor speed;;7;7;RWW;1;-1;-1;-1'; Object Dictionary Item = '6081;Profile Velocity;;7;7;RWW;1;-1;-1;0'; Object Dictionary Item = '6082;End Velocity;0;7;7;RWW;1;-1;-1;0'; Object Dictionary Item = '6083;Profile Acceleration;;7;7;RWW;1;-1;-1;-1'; Object Dictionary Item = '6084;Profile Deceleration;;7;7;RWW;1;-1;-1;-1'; Object Dictionary Item = '6085;Quick Stop Deceleration;;7;7;RW;0;-1;-1;-1'; Object Dictionary Item = '6086;Motion Profile Type;0;3;7;RW;0;-1;-1;-1'; Object Dictionary Item = '6087;Torque Slope;0;7;7;RWW;1;-1;-1;-1'; Object Dictionary Item = '6088;Torque profile type;0;3;7;RW;0;-1;0;0'; Object Dictionary Item = '6089;Position Notation Index;0;2;7;RW;0;-1;127;-128'; Object Dictionary Item = '608A;Position Dimension Index;;5;7;RW;0;-1;255;0'; Object Dictionary Item = '608B;Velocity Notation Index;0;2;7;RW;0;-1;127;-128';
                Object Dictionary Item = '608C;Velocity Dimension Index;;5;7;RW;0;-1;255;0'; Object Dictionary Item = '608D;Acceleration Notation Index;;2;7;RW;0;-1;127;-128'; Object Dictionary Item = '608E;Acceleration Dimension Index;;5;7;RW;0;-1;255;0'; Object Dictionary Item = '608F;Position Encoder Resolution;;-1;8;;-1;3;-1;-1'; Object Dictionary Item = '608Fsub0;Number of entries;2;5;7;RO;0;-1;2;2'; Object Dictionary Item = '608Fsub1;Encoder Increments;1;7;7;RW;0;-1;2147483647;1'; Object Dictionary Item = '608Fsub2;Motor Revolutions;1;7;7;RW;0;-1;16383;1'; Object Dictionary Item = '6090;Velocity Encoder Resolution;;-1;8;;-1;3;-1;-1'; Object Dictionary Item = '6090sub0;Number of entries;2;5;7;RO;0;-1;2;2'; Object Dictionary Item = '6090sub1;Encoder increments per second;1;7;7;RW;0;-1;2147483647;1'; Object Dictionary Item = '6090sub2;Motor revolutions per second;1;7;7;RW;0;-1;16383;1'; Object Dictionary Item = '6093;Position Factor;;-1;8;;-1;3;-1;-1'; Object Dictionary Item = '6093sub0;Number of Entries;2;5;7;RO;0;-1;2;2'; Object Dictionary Item = '6093sub1;Numerator;1;7;7;RW;0;-1;2147483647;1'; Object Dictionary Item = '6093sub2;Feed Constant;1;7;7;RW;0;-1;16383;1'; Object Dictionary Item = '6094;Velocity Encoder Factor;;-1;8;;-1;3;-1;-1'; Object Dictionary Item = '6094sub0;Number of Entries;2;5;7;RO;0;-1;2;2'; Object Dictionary Item = '6094sub1;Numerator;1;7;7;RW;0;-1;2147483647;1'; Object Dictionary Item = '6094sub2;Divisor;1;7;7;RW;0;-1;16383;1'; Object Dictionary Item = '6095;Velocity Factor 1;;-1;8;;-1;3;-1;-1'; Object Dictionary Item = '6095sub0;Number of Entries;2;5;7;RO;0;-1;2;2'; Object Dictionary Item = '6095sub1;Numerator;1;7;7;RW;0;-1;2147483647;1'; Object Dictionary Item = '6095sub2;Divisor;1;7;7;RW;0;-1;16383;1'; Object Dictionary Item = '6096;Velocity Factor 2;;-1;8;;-1;3;-1;-1'; Object Dictionary Item = '6096sub0;Mumber of Entries;2;5;7;RO;0;-1;2;2'; Object Dictionary Item = '6096sub1;Numerator;1;7;7;RW;0;-1;2147483647;1'; Object Dictionary Item = '6096sub2;Divisor;1;7;7;RW;0;-1;16383;1'; Object Dictionary Item = '6097;Acceleration Factor;;-1;8;;-1;3;-1;-1'; Object Dictionary Item = '6097sub0;Number of Entries;2;5;7;RO;0;-1;2;2'; Object Dictionary Item = '6097sub1;Numerator;1;7;7;RW;0;-1;2147483647;1'; Object Dictionary Item = '6097sub2;Divisor;1;7;7;RW;0;-1;16383;1'; Object Dictionary Item = '6098;Homing method;0;2;7;RW;0;-1;35;0'; Object Dictionary Item = '6099;Homing speed;;-1;8;;-1;3;-1;-1'; Object Dictionary Item = '6099sub0;Number of entries;2;5;7;RO;0;-1;2;2'; Object Dictionary Item = '6099sub1;Speed during search for a switch;0;7;7;RW;0;-1;-1;0'; Object Dictionary Item = '6099sub2;Speed during search for an index;0;7;7;RW;0;-1;-1;0'; Object Dictionary Item = '609A;Homing acceleration;;7;7;RW;0;-1;-1;0'; Object Dictionary Item = '60FC;Position Demand Value;;4;7;RO;1;-1;-1;-1'; Object Dictionary Item = '60FD;Digital inputs;0;7;7;RO;1;-1;-1;-1'; Object Dictionary Item = '60FF;Target Velocity;;4;7;RWW;1;-1;2147483647;-2147483648';
                Object Dictionary Item = '6502;Supported drive modes;0x5D;7;7;RO;0;-1;-1;-1'
              output Application.MaxMotorSpeed : UDINT  // Max motor speed
              input  Application.ActVel_RR : DINT  // Velocity actual value
              unmapped channels: Controlword, Target Velocity, Modes of operation, Target Position, Statusword, FaultCode1, WorkState1, Modes Of Operation Display, Position Actual Value
            Rr_Wheel : Axis_CO, Inovance, order no. 0, version 3.5.6.0
                settings: wDriveID = 2; dwRatioTechUnitsDenom = 10; ScalingIncs = 16#1; ScalingMotorTurns2 = 10; LogicId = 0; AdrOffset_8010 = 240; BitOffset_8010 = 0; BitLength_8010 = 16; Address_ = '%QW120'; TYPE_ = 'UINT'; Address_Pointer = ADR(%QW120); AdrOffset_8020 = 248; BitOffset_8020 = 0; BitLength_8020 = 8; Address_ = '%QB248'; TYPE_ = 'SINT'; Address_Pointer = ADR(%QB248); AdrOffset_8030 = 252; BitOffset_8030 = 0; BitLength_8030 = 32; Address_ = '%QD63'; TYPE_ = 'DINT'; Address_Pointer = ADR(%QD63); AdrOffset_8040 = 244; BitOffset_8040 = 0; BitLength_8040 = 32; Address_ = '%QD61'; TYPE_ = 'DINT'; Address_Pointer = ADR(%QD61); AdrOffset_8050 = 0; BitOffset_8050 = 0; BitLength_8050 = 0; Address_ = ''; TYPE_ = ''; Address_Pointer = 0; AdrOffset_8060 = 0; BitOffset_8060 = 0; BitLength_8060 = 0; Address_ = ''; TYPE_ = '';
                  Address_Pointer = 0; AdrOffset_8070 = 0; BitOffset_8070 = 0; BitLength_8070 = 0; Address_ = ''; TYPE_ = ''; Address_Pointer = 0; AdrOffset_8080 = 0; BitOffset_8080 = 0; BitLength_8080 = 0; Address_ = ''; TYPE_ = ''; Address_Pointer = 0; AdrOffset_8510 = 240; BitOffset_8510 = 0; BitLength_8510 = 16; Address_ = '%IW120'; TYPE_ = 'UINT'; Address_Pointer = ADR(%IW120); AdrOffset_8520 = 248; BitOffset_8520 = 0; BitLength_8520 = 32; Address_ = '%ID62'; TYPE_ = 'DINT'; Address_Pointer = ADR(%ID62); AdrOffset_8530 = 246; BitOffset_8530 = 0; BitLength_8530 = 8; Address_ = '%IB246'; TYPE_ = 'SINT'; Address_Pointer = ADR(%IB246); AdrOffset_8540 = 0; BitOffset_8540 = 0; BitLength_8540 = 0; Address_ = ''; TYPE_ = ''; Address_Pointer = 0; AdrOffset_8550 = 0; BitOffset_8550 = 0; BitLength_8550 = 32;
                  Address_ = 'ActVel_RR'; TYPE_ = 'DINT'; Address_Pointer = ADR(ActVel_RR); AdrOffset_8560 = 0; BitOffset_8560 = 0; BitLength_8560 = 0; Address_ = ''; TYPE_ = ''; Address_Pointer = 0; AdrOffset_8570 = 0; BitOffset_8570 = 0; BitLength_8570 = 0; Address_ = ''; TYPE_ = ''; Address_Pointer = 0; Automatic Mapping = True; Slave ID = 2
          FDKServo_PMSM_2 : CANopen Slaver, Inovance, order no. 1525, version 00.00.00.10
              settings: EnableExpertSettings = 1; Error Control.SlaveHeartbeat.ProduceTime = 300; Error Control.SlaveHeartbeat.NrofConsumer = 1; DeviceType = 131474; VendorID = 1459275; ProductNumber = 66128; NrofRxPDO = 4; ValidRxPDO = 15; PdoCommuIndex = 5120; CanId = 513; TxType = 255;  = 3;  = 1614807056;  = 1627324448;  = 1616904200; PdoCommuIndex = 5121; CanId = 769; TxType = 255;  = 2;  = 1618608160;  = 1619001376; PdoCommuIndex = 5122; CanId = 1025; TxType = 255;  = 1; RxPDOMappingArray7.RxPDOMappingArray7 = 1619066912; PdoCommuIndex = 5123; CanId = 1281; TxType = 255;  = 0; NrofTxPDO = 4; ValidTxPDO = 15; PdoCommuIndex = 6144; CanId = 385; TxType = 255; InhibitTime = 100; EventTime = 10;  = 4;  = 1614872592;  = 536870928;
                 = 536936464;  = 1616969736; PdoCommuIndex = 6145; CanId = 641; TxType = 255; InhibitTime = 100; EventTime = 10;  = 2;  = 1617166368;  = 1617690656; PdoCommuIndex = 6146; CanId = 897; TxType = 255; InhibitTime = 100; EventTime = 10;  = 0; PdoCommuIndex = 6147; CanId = 1153; TxType = 255; InhibitTime = 100; EventTime = 10;  = 0; SdoTimeout = 1000; NrofSDO = 65; SdoCommParam = 268763168; SdoCommValue = 128; SdoCommParam = 269877536; SdoCommParam = 269942800; SdoCommValue = 300; SdoCommParam = 269746208; SdoCommValue = 2147483777; SdoCommParam = 269746208; SdoCommValue = 129; SdoCommParam = 335544608; SdoCommValue = 2147484161; SdoCommParam = 335544840; SdoCommValue = 255; SdoCommParam = 369098760; SdoCommParam = 369099040; SdoCommValue = 1614807056;
                SdoCommParam = 369099296; SdoCommValue = 1627324448; SdoCommParam = 369099552; SdoCommValue = 1616904200; SdoCommParam = 369098760; SdoCommValue = 3; SdoCommParam = 335544608; SdoCommValue = 513; SdoCommParam = 335610144; SdoCommValue = 2147484417; SdoCommParam = 335610376; SdoCommValue = 255; SdoCommParam = 369164296; SdoCommParam = 369164576; SdoCommValue = 1618608160; SdoCommParam = 369164832; SdoCommValue = 1619001376; SdoCommParam = 369164296; SdoCommValue = 2; SdoCommParam = 335610144; SdoCommValue = 769; SdoCommParam = 335675680; SdoCommValue = 2147484673; SdoCommParam = 335675912; SdoCommValue = 255; SdoCommParam = 369229832; SdoCommParam = 369230112; SdoCommValue = 1619066912; SdoCommParam = 369229832; SdoCommValue = 1; SdoCommParam = 335675680; SdoCommValue = 1025; SdoCommParam = 335741216; SdoCommValue = 2147484929; SdoCommParam = 335741448; SdoCommValue = 255; SdoCommParam = 369295368; SdoCommParam = 369295368; SdoCommParam = 335741216; SdoCommValue = 1281;
                SdoCommParam = 402653472; SdoCommValue = 2147484033; SdoCommParam = 402653704; SdoCommValue = 255; SdoCommParam = 402653968; SdoCommValue = 100; SdoCommParam = 402654480; SdoCommValue = 10; SdoCommParam = 436207624; SdoCommParam = 436207904; SdoCommValue = 1614872592; SdoCommParam = 436208160; SdoCommValue = 536870928; SdoCommParam = 436208416; SdoCommValue = 536936464; SdoCommParam = 436208672; SdoCommValue = 1616969736; SdoCommParam = 436207624; SdoCommValue = 4; SdoCommParam = 402653472; SdoCommValue = 385; SdoCommParam = 402719008; SdoCommValue = 2147484289; SdoCommParam = 402719240; SdoCommValue = 255; SdoCommParam = 402719504; SdoCommValue = 100; SdoCommParam = 402720016; SdoCommValue = 10; SdoCommParam = 436273160; SdoCommParam = 436273440; SdoCommValue = 1617166368; SdoCommParam = 436273696; SdoCommValue = 1617690656; SdoCommParam = 436273160; SdoCommValue = 2; SdoCommParam = 402719008; SdoCommValue = 641; SdoCommParam = 402784544; SdoCommValue = 2147484545;
                SdoCommParam = 402784776; SdoCommValue = 255; SdoCommParam = 402785040; SdoCommValue = 100; SdoCommParam = 402785552; SdoCommValue = 10; SdoCommParam = 436338696; SdoCommParam = 436338696; SdoCommParam = 402784544; SdoCommValue = 897; SdoCommParam = 402850080; SdoCommValue = 2147484801; SdoCommParam = 402850312; SdoCommValue = 255; SdoCommParam = 402850576; SdoCommValue = 100; SdoCommParam = 402851088; SdoCommValue = 10; SdoCommParam = 436404232; SdoCommParam = 436404232; SdoCommParam = 402850080; SdoCommValue = 1153; FileName = 'FDK_PMSM.eds'; FileVersion = '0x01'; FileRevision = '0x01'; EDSVersion = '4.0'; Description = 'EDS for FDK_Single_DRIVER'; EDS File Path = 'D:\Asoftware\InoProShop\CODESYS\Common\AM600 Data\EdsFile\FDK_PMSM_SIEMENS-VSXXDXX-A-20240203.eds'; EDSVersion = 'FDK, INC.'; VendorNumber = 1459275; ProductName = 'FDKServo-PMSM'; ProductNumber = 66128; RevisionNumber = 0; OrderCode = 'DVPCOPM-SL'; Baudrate = 503; SimpleBootUpSlave = 1; Granularity = 8; DynamicChannelsSupported = 0; GroupMessaging = 0; NrOfRXPDO = 4;
                NrOfTXPDO = 4; LSS_Supported = 1; DummyUsage = 0; SDOType = 0; SDOName = 'Disable COB-ID sync'; SDOType = 0; SDOName = 'Set Heartbeat Consumer'; SDOType = 0; SDOName = 'Set Heartbeat Producer'; SDOType = 0; SDOName = 'Disable Emcy COB-ID'; SDOType = 0; SDOName = 'Set Emcy COB-ID'; SDOType = 0; SDOName = 'Disable PDO'; SDOType = 0; SDOName = 'Set transmission type'; SDOType = 0; SDOName = 'Clear PDO mapping'; SDOType = 0; SDOName = 'Set mapping'; SDOType = 0; SDOName = 'Set mapping'; SDOType = 0; SDOName = 'Set mapping'; SDOType = 0; SDOName = 'Set number of pdos'; SDOType = 0; SDOName = 'Set and enable COB-ID'; SDOType = 0; SDOName = 'Disable PDO'; SDOType = 0; SDOName = 'Set transmission type'; SDOType = 0; SDOName = 'Clear PDO mapping'; SDOType = 0; SDOName = 'Set mapping'; SDOType = 0; SDOName = 'Set mapping'; SDOType = 0;
                SDOName = 'Set number of pdos'; SDOType = 0; SDOName = 'Set and enable COB-ID'; SDOType = 0; SDOName = 'Disable PDO'; SDOType = 0; SDOName = 'Set transmission type'; SDOType = 0; SDOName = 'Clear PDO mapping'; SDOType = 0; SDOName = 'Set mapping'; SDOType = 0; SDOName = 'Set number of pdos'; SDOType = 0; SDOName = 'Set and enable COB-ID'; SDOType = 0; SDOName = 'Disable PDO'; SDOType = 0; SDOName = 'Set transmission type'; SDOType = 0; SDOName = 'Clear PDO mapping'; SDOType = 0; SDOName = 'Set number of pdos'; SDOType = 0; SDOName = 'Set and enable COB-ID'; SDOType = 0; SDOName = 'Disable PDO'; SDOType = 0; SDOName = 'Set transmission type'; SDOType = 0; SDOName = 'Set inhibit time'; SDOType = 0; SDOName = 'Set event time'; SDOType = 0; SDOName = 'Clear PDO mapping'; SDOType = 0; SDOName = 'Set mapping'; SDOType = 0; SDOName = 'Set mapping'; SDOType = 0;
                SDOName = 'Set mapping'; SDOType = 0; SDOName = 'Set mapping'; SDOType = 0; SDOName = 'Set number of pdos'; SDOType = 0; SDOName = 'Set and enable COB-ID'; SDOType = 0; SDOName = 'Disable PDO'; SDOType = 0; SDOName = 'Set transmission type'; SDOType = 0; SDOName = 'Set inhibit time'; SDOType = 0; SDOName = 'Set event time'; SDOType = 0; SDOName = 'Clear PDO mapping'; SDOType = 0; SDOName = 'Set mapping'; SDOType = 0; SDOName = 'Set mapping'; SDOType = 0; SDOName = 'Set number of pdos'; SDOType = 0; SDOName = 'Set and enable COB-ID'; SDOType = 0; SDOName = 'Disable PDO'; SDOType = 0; SDOName = 'Set transmission type'; SDOType = 0; SDOName = 'Set inhibit time'; SDOType = 0; SDOName = 'Set event time'; SDOType = 0; SDOName = 'Clear PDO mapping'; SDOType = 0; SDOName = 'Set number of pdos'; SDOType = 0; SDOName = 'Set and enable COB-ID'; SDOType = 0;
                SDOName = 'Disable PDO'; SDOType = 0; SDOName = 'Set transmission type'; SDOType = 0; SDOName = 'Set inhibit time'; SDOType = 0; SDOName = 'Set event time'; SDOType = 0; SDOName = 'Clear PDO mapping'; SDOType = 0; SDOName = 'Set number of pdos'; SDOType = 0; SDOName = 'Set and enable COB-ID'; Recv PDO Mapping Name.Recv PDO Mapping Name = 'Controlword'; Recv PDO Mapping Name.Recv PDO Mapping Name = 'Target Velocity'; Recv PDO Mapping Name.Recv PDO Mapping Name = 'Modes of operation'; Recv PDO Mapping Name.Recv PDO Mapping Name = 'Target Position'; Recv PDO Mapping Name.Recv PDO Mapping Name = 'Max motor speed'; Recv PDO Mapping Name.Recv PDO Mapping Name = 'Profile Velocity'; Send PDO Mapping Name.Send PDO Mapping Name = 'Statusword'; Send PDO Mapping Name.Send PDO Mapping Name = 'FaultCode1'; Send PDO Mapping Name.Send PDO Mapping Name = 'WorkState1'; Send PDO Mapping Name.Send PDO Mapping Name = 'Modes Of Operation Display'; Send PDO Mapping Name.Send PDO Mapping Name = 'Position Actual Value'; Send PDO Mapping Name.Send PDO Mapping Name = 'Velocity actual value'; Is Manual change COB-ID = 0; Is Manual change COB-ID = 0; Is Manual change COB-ID = 0; Is Manual change COB-ID = 0; Is Manual change COB-ID = 0; Is Manual change COB-ID = 0; Is Manual change COB-ID = 0; Is Manual change COB-ID = 0; MandatoryObjs = 3; Object Dictionary Item = '1000;CAN Controller Type;0x20192;7;7;RO;0;-1;-1;-1'; Object Dictionary Item = '1001;Error Register;0;5;7;RO;0;-1;-1;-1'; Object Dictionary Item = '1018;Identity Object;;-1;9;;-1;4;-1;-1'; Object Dictionary Item = '1018sub0;number of entries;3;5;7;RO;0;-1;4;1'; Object Dictionary Item = '1018sub1;Vendor ID;0x0016444B;7;7;RO;0;-1;-1;-1'; Object Dictionary Item = '1018sub2;Product code;0x00010250;7;7;RO;0;-1;-1;-1';
                Object Dictionary Item = '1018sub3;Revision number;0x00000000;7;7;RO;0;-1;-1;-1'; ManufacturerObjs = 30; Object Dictionary Item = '2000;FaultCode1;;6;7;RO;1;-1;65535;0'; Object Dictionary Item = '2001;WorkState1;;6;7;RO;1;-1;65535;0'; Object Dictionary Item = '2002;Motor_T;;6;7;RO;1;-1;-1;-1'; Object Dictionary Item = '2004;WARN;;6;7;RO;1;-1;65535;0'; Object Dictionary Item = '2005;CurrentBase;;6;7;RO;1;-1;65535;0'; Object Dictionary Item = '2006;LineEncoder;;4;7;RO;1;-1;65535;0'; Object Dictionary Item = '2007;Feedback Type;;6;7;RW;0;-1;65535;0'; Object Dictionary Item = '2008;Pole Pairs;;6;7;RW;0;-1;65535;0'; Object Dictionary Item = '2009;CAN ID;;5;7;RW;0;-1;-1;-1'; Object Dictionary Item = '200A;Can Baud Rate;;6;7;RW;0;-1;-1;-1'; Object Dictionary Item = '200B;Rated Current;;3;7;RW;0;-1;-1;-1'; Object Dictionary Item = '200C;Rated Speed;;3;7;RW;0;-1;-1;-1'; Object Dictionary Item = '200D;Overload Current;;6;7;RW;1;-1;-1;-1'; Object Dictionary Item = '200E;Overload Time;;6;7;RW;1;-1;-1;-1'; Object Dictionary Item = '200F;Current Loop P;;6;7;RW;1;-1;-1;-1'; Object Dictionary Item = '2010;Current Loop I;;6;7;RW;1;-1;-1;-1'; Object Dictionary Item = '2011;Speed Loop p0;;6;7;RW;1;-1;-1;-1'; Object Dictionary Item = '2012;Speed Loop P1;;6;7;RW;1;-1;-1;-1'; Object Dictionary Item = '2013;Speed Loop I;;6;7;RW;1;-1;-1;-1'; Object Dictionary Item = '2014;Position Loop P0;;6;7;RW;1;-1;-1;-1'; Object Dictionary Item = '2015;Position Loop P1;;6;7;RW;1;-1;-1;-1'; Object Dictionary Item = '2016;Command0;;6;7;RW;1;-1;-1;-1'; Object Dictionary Item = '2017;Command1;;6;7;RW;1;-1;-1;-1'; Object Dictionary Item = '2018;Software Limited Cache;;6;7;RW;1;-1;-1;-1'; Object Dictionary Item = '2019;Software Limited Forward Position;;4;7;RW;1;-1;-1;-1'; Object Dictionary Item = '201A;Software Limited Reverse Position;;4;7;RW;1;-1;-1;-1'; Object Dictionary Item = '201B;RS485_NodeID;;6;7;RW;1;-1;-1;-1'; Object Dictionary Item = '201C;RS485_Baudrate;;6;7;RW;1;-1;-1;-1'; Object Dictionary Item = '201D;RS485_Protocol;;6;7;RW;1;-1;-1;-1'; Object Dictionary Item = '22A2;System_T;;6;7;RO;1;-1;-1;-1'; OptionsObjs = 104; Object Dictionary Item = '1002;Manufacturer Status Register;;7;7;RO;1;-1;-1;-1'; Object Dictionary Item = '1003;Pre-defined Error Field;;-1;8;;-1;17;-1;-1'; Object Dictionary Item = '1003sub0;Number of Errors;0;5;7;RW;0;-1;16;0'; Object Dictionary Item = '1003sub1;Standard Error Field;0;7;7;RO;0;-1;-1;0'; Object Dictionary Item = '1003sub2;Standard Error Field;0;7;7;RO;0;-1;-1;0'; Object Dictionary Item = '1003sub3;Standard Error Field;0;7;7;RO;0;-1;-1;0'; Object Dictionary Item = '1003sub4;Standard Error Field;0;7;7;RO;0;-1;-1;0';
                Object Dictionary Item = '1003sub5;Standard Error Field;0;7;7;RO;0;-1;-1;0'; Object Dictionary Item = '1003sub6;Standard Error Field;0;7;7;RO;0;-1;-1;0'; Object Dictionary Item = '1003sub7;Standard Error Field;0;7;7;RO;0;-1;-1;0'; Object Dictionary Item = '1003sub8;Standard Error Field;0;7;7;RO;0;-1;-1;0'; Object Dictionary Item = '1003sub9;Standard Error Field;0;7;7;RO;0;-1;-1;0'; Object Dictionary Item = '1003suba;Standard Error Field;0;7;7;RO;0;-1;-1;0'; Object Dictionary Item = '1003subb;Standard Error Field;0;7;7;RO;0;-1;-1;0'; Object Dictionary Item = '1003subc;Standard Error Field;0;7;7;RO;0;-1;-1;0'; Object Dictionary Item = '1003subd;Standard Error Field;0;7;7;RO;0;-1;-1;0'; Object Dictionary Item = '1003sube;Standard Error Field;0;7;7;RO;0;-1;-1;0'; Object Dictionary Item = '1003subf;Standard Error Field;0;7;7;RO;0;-1;-1;0'; Object Dictionary Item = '1003sub10;Standard Error Field;0;7;7;RO;0;-1;-1;0'; Object Dictionary Item = '1005;COB-ID SYNC-message;0x80;7;7;RW;0;-1;-1;-1'; Object Dictionary Item = '1006;Communication Cycle Period;0;7;7;RW;0;-1;-1;0'; Object Dictionary Item = '1008;Manufacturer Device Name;;9;7;CONST;0;-1;-1;-1'; Object Dictionary Item = '1009;Manufacturer Hardware Version;;9;7;CONST;0;-1;-1;-1'; Object Dictionary Item = '100A;Manufacturer Software Version;;9;7;CONST;0;-1;-1;-1'; Object Dictionary Item = '100B;Node-ID;1;5;7;RO;0;-1;127;1'; Object Dictionary Item = '1010;Store Parameters;;-1;8;;-1;4;-1;-1'; Object Dictionary Item = '1010sub0;Largest Supported Sub-index;3;5;7;RO;0;-1;3;3'; Object Dictionary Item = '1010sub1;Save All Parameters;;7;7;RW;0;-1;-1;-1'; Object Dictionary Item = '1010sub2;Save Communication Parameters;0;7;7;RW;0;-1;-1;-1'; Object Dictionary Item = '1010sub3;Save ApplicationParameters;0;7;7;RW;0;-1;-1;-1'; Object Dictionary Item = '1011;Restore  Parameters;;-1;8;;-1;4;-1;-1'; Object Dictionary Item = '1011sub0;Largest Supported Sub-index;3;5;7;RO;0;-1;3;3'; Object Dictionary Item = '1011sub1;Restore All Parameters;;7;7;RW;0;-1;-1;-1'; Object Dictionary Item = '1011sub2;Restore Communication Parameters;0;7;7;RW;0;-1;-1;-1'; Object Dictionary Item = '1011sub3;Restore ApplicationParameters;0;7;7;RW;0;-1;-1;-1'; Object Dictionary Item = '1012;COB-ID Time Stamp Message;0x80000100;7;7;RW;0;-1;-1;-1'; Object Dictionary Item = '1013;High Resolution TimeStamp;0;7;7;RW;0;-1;-1;0'; Object Dictionary Item = '1014;COB-ID Emergency Message;$NODEID+0x80;7;7;RW;0;-1;-1;-1'; Object Dictionary Item = '1016;Consumer Heartbeat Time;;-1;8;;-1;2;-1;-1'; Object Dictionary Item = '1016sub0;Number of Entries;1;5;7;RO;0;-1;1;1'; Object Dictionary Item = '1016sub1;Consumer Heartbeat Time;0;7;7;RW;0;-1;-1;-1'; Object Dictionary Item = '1017;Producer heartbeat time;0;6;7;RW;0;-1;-1;-1'; Object Dictionary Item = '1023;OS Command;;-1;9;;-1;4;-1;-1'; Object Dictionary Item = '1023sub0;Number of Entries;3;5;7;RO;0;-1;3;3'; Object Dictionary Item = '1023sub1;Command;;10;7;WO;0;-1;-1;-1'; Object Dictionary Item = '1023sub2;Status;0;5;7;RO;0;-1;255;0'; Object Dictionary Item = '1023sub3;Reply;;10;7;RO;0;-1;-1;-1';
                Object Dictionary Item = '1024;OS Command Mode;0;5;7;WO;0;-1;-1;-1'; Object Dictionary Item = '1029;Error Behavior;;-1;8;;-1;2;-1;-1'; Object Dictionary Item = '1029sub0;Number of Error Classes;1;5;7;RO;0;-1;1;1'; Object Dictionary Item = '1029sub1;Communication Error;1;5;7;RW;0;-1;2;0'; Object Dictionary Item = '1200;1st Server SDO Parameter;;-1;9;;-1;3;-1;-1'; Object Dictionary Item = '1200sub0;Number of Entries;2;5;7;RO;0;-1;2;2'; Object Dictionary Item = '1200sub1;COB-ID Client->Server (Rx);$NODEID+0x600;7;7;RO;0;-1;-1;-1'; Object Dictionary Item = '1200sub2;COB-ID Server ->Client (Tx);$NODEID+0x580;7;7;RO;0;-1;-1;-1'; Object Dictionary Item = '1400;1st Receive PDO Parameter;;-1;9;;-1;3;-1;-1'; Object Dictionary Item = '1400sub0;Largest Sub-Index Supported;2;5;7;RO;0;-1;2;2'; Object Dictionary Item = '1400sub1;COB-ID Used by PDO;$NODEID+0x200;7;7;RW;0;-1;-1;-1'; Object Dictionary Item = '1400sub2;Transmission Type;0xFF;5;7;RW;0;-1;255;0'; Object Dictionary Item = '1600;1st Receive PDO Mapping;;-1;9;;-1;5;-1;-1'; Object Dictionary Item = '1600sub0;Number of Mapped Application Objects in PDO;3;5;7;RW;0;-1;8;0'; Object Dictionary Item = '1600sub1;PDO Mapping for the 1st Application Object to Be Mapped;0x60400010;7;7;RW;0;-1;-1;-1'; Object Dictionary Item = '1600sub2;PDO Mapping for the 2nd Application Object to Be Mapped;0x60FF0020;7;7;RW;0;-1;-1;-1'; Object Dictionary Item = '1600sub3;PDO Mapping for the 3rd Application Object to Be Mapped;0x60600008;7;7;RW;0;-1;-1;-1'; Object Dictionary Item = '1600sub4;PDO Mapping for the 4th Application Object to Be Mapped;;7;7;RW;0;-1;-1;-1'; Object Dictionary Item = '1401;2nd Receive PDO parameter;;-1;9;;-1;3;-1;-1'; Object Dictionary Item = '1401sub0;Number of Entries;2;5;7;RO;0;-1;2;2'; Object Dictionary Item = '1401sub1;COB-ID used by PDO;$NODEID+0x300;7;7;RW;0;-1;-1;-1'; Object Dictionary Item = '1401sub2;Transmission Type;0xFF;5;7;RW;0;-1;255;0'; Object Dictionary Item = '1601;2nd Receive PDO Mapping;;-1;9;;-1;5;-1;-1'; Object Dictionary Item = '1601sub0;Number of Mapped Application Objects in PDO;2;5;7;RW;0;-1;8;0'; Object Dictionary Item = '1601sub1;PDO Mapping for the 1st Application Object to Be Mapped;0x607A0020;7;7;RW;0;-1;-1;-1'; Object Dictionary Item = '1601sub2;PDO Mapping for the 2nd Application Object to Be Mapped;0x60800020;7;7;RW;0;-1;-1;-1'; Object Dictionary Item = '1601sub3;PDO Mapping for the 3rd Application Object to Be Mapped;;7;7;RW;0;-1;-1;-1'; Object Dictionary Item = '1601sub4;PDO Mapping for the 4th Application Object to Be Mapped;;7;7;RW;0;-1;-1;-1'; Object Dictionary Item = '1402;3rd Receive PDO Parameters;;-1;9;;-1;3;-1;-1'; Object Dictionary Item = '1402sub0;number of elements;2;5;7;RO;0;-1;2;2'; Object Dictionary Item = '1402sub1;COB-ID used by PDO;$NODEID+0x400;7;7;RW;0;-1;-1;-1'; Object Dictionary Item = '1402sub2;Transmission Type;0xFF;5;7;RW;0;-1;255;0'; Object Dictionary Item = '1602;3rd Receive PDO Mapping;;-1;9;;-1;5;-1;-1'; Object Dictionary Item = '1602sub0;Number of Mapped Application Objects in PDO;0;5;7;RW;0;-1;8;0'; Object Dictionary Item = '1602sub1;PDO Mapping for the 1st Application Object to Be Mapped;;7;7;RW;0;-1;-1;-1'; Object Dictionary Item = '1602sub2;PDO Mapping for the 2nd Application Object to Be Mapped;;7;7;RW;0;-1;-1;-1'; Object Dictionary Item = '1602sub3;PDO Mapping for the 3rd Application Object to Be Mapped;;7;7;RW;0;-1;-1;-1'; Object Dictionary Item = '1602sub4;PDO Mapping for the 4th Application Object to Be Mapped;;7;7;RW;0;-1;-1;-1'; Object Dictionary Item = '1403;4th Received PDO Parameters;;-1;9;;-1;3;-1;-1'; Object Dictionary Item = '1403sub0;number of elements;2;5;7;RO;0;-1;2;2';
                Object Dictionary Item = '1403sub1;COB-ID used by PDO;$NODEID+0x500;7;7;RW;0;-1;-1;-1'; Object Dictionary Item = '1403sub2;Transmission Type;0xFF;5;7;RW;0;-1;255;0'; Object Dictionary Item = '1603;4th Receive PDO Mapping;;-1;9;;-1;5;-1;-1'; Object Dictionary Item = '1603sub0;Number of Mapped Application Objects in PDO;0;5;7;RW;0;-1;8;0'; Object Dictionary Item = '1603sub1;PDO Mapping for the 1st Application Object to Be Mapped;;7;7;RW;0;-1;-1;-1'; Object Dictionary Item = '1603sub2;PDO Mapping for the 2nd Application Object to Be Mapped;;7;7;RW;0;-1;-1;-1'; Object Dictionary Item = '1603sub3;PDO Mapping for the 3rd Application Object to Be Mapped;;7;7;RW;0;-1;-1;-1'; Object Dictionary Item = '1603sub4;PDO Mapping for the 4th Application Object to Be Mapped;;7;7;RW;0;-1;-1;-1'; Object Dictionary Item = '1800;1st Transmit PDO Parameter;;-1;9;;-1;6;-1;-1'; Object Dictionary Item = '1800sub0;Largest Sub-Index Supported;5;5;7;RO;0;-1;5;5'; Object Dictionary Item = '1800sub1;COB-ID Used by PDO;$NODEID+0x00000180;7;7;RW;0;-1;-1;-1'; Object Dictionary Item = '1800sub2;Transmission Type;255;5;7;RW;0;-1;255;0'; Object Dictionary Item = '1800sub3;Inhibit Time;100;6;7;RW;0;-1;-1;-1'; Object Dictionary Item = '1800sub4;Reserved;;5;7;RW;0;-1;-1;-1'; Object Dictionary Item = '1800sub5;Event Timer;10;6;7;RW;0;-1;-1;-1'; Object Dictionary Item = '1A00;1st Transmit PDO Mapping;;-1;9;;-1;5;-1;-1'; Object Dictionary Item = '1A00sub0;Number Of Mapped Application Object In PDO.;4;5;7;RW;0;-1;8;0'; Object Dictionary Item = '1A00sub1;PDO Mapping For The 1st Application Object To Be Mapped;0x60410010;7;7;RW;0;-1;-1;-1'; Object Dictionary Item = '1A00sub2;PDO Mapping For The 2nd  Application Object To Be Mapped;0x20000010;7;7;RW;0;-1;-1;-1'; Object Dictionary Item = '1A00sub3;PDO Mapping For The 3rd Application Object To Be Mapped;0x20010010;7;7;RW;0;-1;-1;-1'; Object Dictionary Item = '1A00sub4;PDO Mapping For The 4th Application Object To Be Mapped;0x60610008;7;7;RW;0;-1;-1;-1'; Object Dictionary Item = '1801;2nd Transmit PDO Parameter;;-1;9;;-1;6;-1;-1'; Object Dictionary Item = '1801sub0;Largest Sub-Index Supported;5;5;7;RO;0;-1;5;5'; Object Dictionary Item = '1801sub1;COB-ID Used  by PDO;$NODEID+0x00000280;7;7;RW;0;-1;-1;-1'; Object Dictionary Item = '1801sub2;Transmission Type;255;5;7;RW;0;-1;255;0'; Object Dictionary Item = '1801sub3;Inhibit Time;100;6;7;RW;0;-1;-1;-1'; Object Dictionary Item = '1801sub4;Reserved;;5;7;RW;0;-1;-1;-1'; Object Dictionary Item = '1801sub5;Event Timer;10;6;7;RW;0;-1;-1;-1'; Object Dictionary Item = '1A01;2nd Transmit PDO Mapping;;-1;9;;-1;5;-1;-1'; Object Dictionary Item = '1A01sub0;Number Of Mapped Application Object In PDO.;2;5;7;RW;0;-1;8;0'; Object Dictionary Item = '1A01sub1;PDO Mapping For The 1st Application Object To Be Mapped;0x60640020;7;7;RW;0;-1;-1;-1'; Object Dictionary Item = '1A01sub2;PDO Mapping For The 2nd  Application Object To Be Mapped;0x606C0020;7;7;RW;0;-1;-1;-1'; Object Dictionary Item = '1A01sub3;PDO Mapping For The 3rd Application Object To Be Mapped;;7;7;RW;0;-1;-1;-1'; Object Dictionary Item = '1A01sub4;PDO Mapping For The 4th Application Object To Be Mapped;;7;7;RW;0;-1;-1;-1'; Object Dictionary Item = '1802;3rd Transmit PDO Parameter;;-1;9;;-1;6;-1;-1'; Object Dictionary Item = '1802sub0;Largest Sub-Index Supported;5;5;7;RO;0;-1;5;5'; Object Dictionary Item = '1802sub1;COB-ID Used  by PDO;$NODEID+0x00000380;7;7;RW;0;-1;-1;-1'; Object Dictionary Item = '1802sub2;Transmission Type;255;5;7;RW;0;-1;255;0'; Object Dictionary Item = '1802sub3;Inhibit Time;100;6;7;RW;0;-1;-1;-1'; Object Dictionary Item = '1802sub4;Reserved;;5;7;RW;0;-1;-1;-1';
                Object Dictionary Item = '1802sub5;Event Timer;10;6;7;RW;0;-1;-1;-1'; Object Dictionary Item = '1A02;3rd Transmit PDO  Mapping;;-1;9;;-1;5;-1;-1'; Object Dictionary Item = '1A02sub0;Number Of Mapped Application Object In PDO.;0;5;7;RW;0;-1;8;0'; Object Dictionary Item = '1A02sub1;PDO Mapping For The 1st Application Object To Be Mapped;;7;7;RW;0;-1;-1;-1'; Object Dictionary Item = '1A02sub2;PDO Mapping For The 2nd Application Object To Be Mapped;;7;7;RW;0;-1;-1;-1'; Object Dictionary Item = '1A02sub3;PDO Mapping For The 3rd Application Object To Be Mapped;;7;7;RW;0;-1;-1;-1'; Object Dictionary Item = '1A02sub4;PDO Mapping For The 4th Application Object To Be Mapped;;7;7;RW;0;-1;-1;-1'; Object Dictionary Item = '1803;4th Transmit PDO Parameter;;-1;9;;-1;6;-1;-1'; Object Dictionary Item = '1803sub0;Largest Sub-Index Supported;5;5;7;RO;0;-1;5;5'; Object Dictionary Item = '1803sub1;COB-ID Used  by PDO;$NODEID+0x00000480;7;7;RW;0;-1;-1;-1'; Object Dictionary Item = '1803sub2;Transmission Type;255;5;7;RW;0;-1;255;0'; Object Dictionary Item = '1803sub3;Inhibit Time;100;6;7;RW;0;-1;-1;-1'; Object Dictionary Item = '1803sub4;Reserved;;5;7;RW;0;-1;-1;-1'; Object Dictionary Item = '1803sub5;Event Timer;10;6;7;RW;0;-1;-1;-1'; Object Dictionary Item = '1A03;4th Transmit PDO  Mapping;;-1;9;;-1;5;-1;-1'; Object Dictionary Item = '1A03sub0;Number Of Mapped Application Object In PDO.;0;5;7;RW;0;-1;8;0'; Object Dictionary Item = '1A03sub1;PDO Mapping For The 1st Application Object To Be Mapped;;7;7;RW;0;-1;-1;-1'; Object Dictionary Item = '1A03sub2;PDO Mapping For The 2nd Application Object To Be Mapped;;7;7;RW;0;-1;-1;-1'; Object Dictionary Item = '1A03sub3;PDO Mapping For The 3rd Application Object To Be Mapped;;7;7;RW;0;-1;-1;-1'; Object Dictionary Item = '1A03sub4;PDO Mapping For The 4th Application Object To Be Mapped;;7;7;RW;0;-1;-1;-1'; Object Dictionary Item = '6007;Abort Connection Option Code;0;3;7;RW;0;-1;32767;-32768'; Object Dictionary Item = '603F;Error code;0;6;7;RO;0;-1;65535;0'; Object Dictionary Item = '6040;Controlword;;6;7;RWW;1;-1;65535;0'; Object Dictionary Item = '6041;Statusword;;6;7;RO;1;-1;65535;0'; Object Dictionary Item = '605A;Quick Stop Option Code;2;3;7;RW;0;-1;6;0'; Object Dictionary Item = '605B;Shutdown Option Code;0;3;7;RW;0;-1;1;0'; Object Dictionary Item = '605C;Disable Operation Option Code;1;3;7;RW;0;-1;1;0'; Object Dictionary Item = '605D;Halt Option Code;1;3;7;RW;0;-1;2;0'; Object Dictionary Item = '605E;Fault Reaction Option Code;0;3;7;RW;0;-1;0;0'; Object Dictionary Item = '6060;Modes of operation;;2;7;RWW;1;-1;7;-1'; Object Dictionary Item = '6061;Modes Of Operation Display;;2;7;RO;1;-1;7;-1'; Object Dictionary Item = '6062;Position Demand Value;0;4;7;RO;1;-1;2147483647;-1'; Object Dictionary Item = '6063;Position Actual Value;;4;7;RO;1;-1;2147483647;-1'; Object Dictionary Item = '6064;Position Actual Value;0;4;7;RO;1;-1;2147483647;-1'; Object Dictionary Item = '6065;Following Error Window;;7;7;RW;0;-1;-1;0'; Object Dictionary Item = '6066;Following Error Time Out;;6;7;RW;0;-1;65535;0'; Object Dictionary Item = '6067;Position Window;;7;7;RW;0;-1;32000;0'; Object Dictionary Item = '6068;Position Windows Time;;6;7;RW;0;-1;100;0'; Object Dictionary Item = '6069;Velocity Sensor Actual Value;;4;7;RO;1;-1;-1;-1'; Object Dictionary Item = '606A;Sensor selection code;;3;7;RW;0;-1;1;0';
                Object Dictionary Item = '606B;Velocity Demand Value;;4;7;RO;1;-1;-1;-1'; Object Dictionary Item = '606C;Velocity actual value;;4;7;RO;1;-1;-1;-1'; Object Dictionary Item = '606D;Velocity Window;;6;7;RW;0;-1;65535;0'; Object Dictionary Item = '606E;Velocity Window Time;;6;7;RW;0;-1;65535;0'; Object Dictionary Item = '606F;Velocity Threshold;;6;7;RW;0;-1;65535;0'; Object Dictionary Item = '6070;Velocity Threshold Time;;6;7;RW;0;-1;65535;0'; Object Dictionary Item = '6071;Target Torque;0;3;7;RWW;1;-1;-1;-1'; Object Dictionary Item = '6072;Max Torque;0;6;7;RW;0;-1;-1;-1'; Object Dictionary Item = '6073;Max Current;0;6;7;RW;0;-1;-1;-1'; Object Dictionary Item = '6074;Torque demand value;0;3;7;RO;1;-1;-1;-1'; Object Dictionary Item = '6075;Motor rated current;0;7;7;RW;0;-1;-1;-1'; Object Dictionary Item = '6076;Motor rated torque;0;7;7;RW;0;-1;-1;-1'; Object Dictionary Item = '6077;Torque actual value;0;3;7;RO;1;-1;-1;-1'; Object Dictionary Item = '6078;Current Actual Value;0;3;7;RO;1;-1;-1;-1'; Object Dictionary Item = '607A;Target Position;;4;7;RWW;1;-1;2147483647;-2147483648'; Object Dictionary Item = '607B;Position Range Limit;;-1;8;;-1;3;-1;-1'; Object Dictionary Item = '607Bsub0;Number of Entries;2;5;7;RO;0;-1;2;2'; Object Dictionary Item = '607Bsub1;Min Position Range Limit;-1000000000;4;7;RW;0;-1;-1;-1'; Object Dictionary Item = '607Bsub2;Max Position Range Limit;1000000000;4;7;RW;0;-1;-1;-1'; Object Dictionary Item = '607C;Home offset;0;4;7;RW;0;-1;2147483647;-2147483648'; Object Dictionary Item = '607D;Software Position Limit;;-1;8;;-1;3;-1;-1'; Object Dictionary Item = '607Dsub0;Number of Entries;2;5;7;RO;0;-1;2;2'; Object Dictionary Item = '607Dsub1;Min Position Limit;-1000000000;4;7;RW;0;-1;-1;-1'; Object Dictionary Item = '607Dsub2;Max Position Limit;1000000000;4;7;RW;0;-1;-1;-1'; Object Dictionary Item = '607E;Polarity;0;5;7;RWW;1;-1;-1;-1'; Object Dictionary Item = '607F;Max Profile Velocity;;7;7;RW;0;-1;-1;0'; Object Dictionary Item = '6080;Max motor speed;;7;7;RWW;1;-1;-1;-1'; Object Dictionary Item = '6081;Profile Velocity;;7;7;RWW;1;-1;-1;0'; Object Dictionary Item = '6082;End Velocity;0;7;7;RWW;1;-1;-1;0'; Object Dictionary Item = '6083;Profile Acceleration;;7;7;RWW;1;-1;-1;-1'; Object Dictionary Item = '6084;Profile Deceleration;;7;7;RWW;1;-1;-1;-1'; Object Dictionary Item = '6085;Quick Stop Deceleration;;7;7;RW;0;-1;-1;-1'; Object Dictionary Item = '6086;Motion Profile Type;0;3;7;RW;0;-1;-1;-1'; Object Dictionary Item = '6087;Torque Slope;0;7;7;RWW;1;-1;-1;-1'; Object Dictionary Item = '6088;Torque profile type;0;3;7;RW;0;-1;0;0'; Object Dictionary Item = '6089;Position Notation Index;0;2;7;RW;0;-1;127;-128'; Object Dictionary Item = '608A;Position Dimension Index;;5;7;RW;0;-1;255;0'; Object Dictionary Item = '608B;Velocity Notation Index;0;2;7;RW;0;-1;127;-128'; Object Dictionary Item = '608C;Velocity Dimension Index;;5;7;RW;0;-1;255;0'; Object Dictionary Item = '608D;Acceleration Notation Index;;2;7;RW;0;-1;127;-128';
                Object Dictionary Item = '608E;Acceleration Dimension Index;;5;7;RW;0;-1;255;0'; Object Dictionary Item = '608F;Position Encoder Resolution;;-1;8;;-1;3;-1;-1'; Object Dictionary Item = '608Fsub0;Number of entries;2;5;7;RO;0;-1;2;2'; Object Dictionary Item = '608Fsub1;Encoder Increments;1;7;7;RW;0;-1;2147483647;1'; Object Dictionary Item = '608Fsub2;Motor Revolutions;1;7;7;RW;0;-1;16383;1'; Object Dictionary Item = '6090;Velocity Encoder Resolution;;-1;8;;-1;3;-1;-1'; Object Dictionary Item = '6090sub0;Number of entries;2;5;7;RO;0;-1;2;2'; Object Dictionary Item = '6090sub1;Encoder increments per second;1;7;7;RW;0;-1;2147483647;1'; Object Dictionary Item = '6090sub2;Motor revolutions per second;1;7;7;RW;0;-1;16383;1'; Object Dictionary Item = '6093;Position Factor;;-1;8;;-1;3;-1;-1'; Object Dictionary Item = '6093sub0;Number of Entries;2;5;7;RO;0;-1;2;2'; Object Dictionary Item = '6093sub1;Numerator;1;7;7;RW;0;-1;2147483647;1'; Object Dictionary Item = '6093sub2;Feed Constant;1;7;7;RW;0;-1;16383;1'; Object Dictionary Item = '6094;Velocity Encoder Factor;;-1;8;;-1;3;-1;-1'; Object Dictionary Item = '6094sub0;Number of Entries;2;5;7;RO;0;-1;2;2'; Object Dictionary Item = '6094sub1;Numerator;1;7;7;RW;0;-1;2147483647;1'; Object Dictionary Item = '6094sub2;Divisor;1;7;7;RW;0;-1;16383;1'; Object Dictionary Item = '6095;Velocity Factor 1;;-1;8;;-1;3;-1;-1'; Object Dictionary Item = '6095sub0;Number of Entries;2;5;7;RO;0;-1;2;2'; Object Dictionary Item = '6095sub1;Numerator;1;7;7;RW;0;-1;2147483647;1'; Object Dictionary Item = '6095sub2;Divisor;1;7;7;RW;0;-1;16383;1'; Object Dictionary Item = '6096;Velocity Factor 2;;-1;8;;-1;3;-1;-1'; Object Dictionary Item = '6096sub0;Mumber of Entries;2;5;7;RO;0;-1;2;2'; Object Dictionary Item = '6096sub1;Numerator;1;7;7;RW;0;-1;2147483647;1'; Object Dictionary Item = '6096sub2;Divisor;1;7;7;RW;0;-1;16383;1'; Object Dictionary Item = '6097;Acceleration Factor;;-1;8;;-1;3;-1;-1'; Object Dictionary Item = '6097sub0;Number of Entries;2;5;7;RO;0;-1;2;2'; Object Dictionary Item = '6097sub1;Numerator;1;7;7;RW;0;-1;2147483647;1'; Object Dictionary Item = '6097sub2;Divisor;1;7;7;RW;0;-1;16383;1'; Object Dictionary Item = '6098;Homing method;0;2;7;RW;0;-1;35;0'; Object Dictionary Item = '6099;Homing speed;;-1;8;;-1;3;-1;-1'; Object Dictionary Item = '6099sub0;Number of entries;2;5;7;RO;0;-1;2;2'; Object Dictionary Item = '6099sub1;Speed during search for a switch;0;7;7;RW;0;-1;-1;0'; Object Dictionary Item = '6099sub2;Speed during search for an index;0;7;7;RW;0;-1;-1;0'; Object Dictionary Item = '609A;Homing acceleration;;7;7;RW;0;-1;-1;0'; Object Dictionary Item = '60FC;Position Demand Value;;4;7;RO;1;-1;-1;-1'; Object Dictionary Item = '60FD;Digital inputs;0;7;7;RO;1;-1;-1;-1'; Object Dictionary Item = '60FF;Target Velocity;;4;7;RWW;1;-1;2147483647;-2147483648'; Object Dictionary Item = '6502;Supported drive modes;0x5D;7;7;RO;0;-1;-1;-1'
              output Application.MaxMotorSpeed : UDINT  // Max motor speed
              input  Application.ActVel_RL : DINT  // Velocity actual value
              unmapped channels: Controlword, Target Velocity, Modes of operation, Target Position, Profile Velocity, Statusword, FaultCode1, WorkState1, Modes Of Operation Display, Position Actual Value
            Rl_Wheel : Axis_CO, Inovance, order no. 0, version 3.5.6.0
                settings: wDriveID = 4; dwRatioTechUnitsDenom = 10; ScalingIncs = 16#1; ScalingMotorTurns2 = 10; LogicId = 0; AdrOffset_8010 = 272; BitOffset_8010 = 0; BitLength_8010 = 16; Address_ = '%QW136'; TYPE_ = 'UINT'; Address_Pointer = ADR(%QW136); AdrOffset_8020 = 280; BitOffset_8020 = 0; BitLength_8020 = 8; Address_ = '%QB280'; TYPE_ = 'SINT'; Address_Pointer = ADR(%QB280); AdrOffset_8030 = 284; BitOffset_8030 = 0; BitLength_8030 = 32; Address_ = '%QD71'; TYPE_ = 'DINT'; Address_Pointer = ADR(%QD71); AdrOffset_8040 = 276; BitOffset_8040 = 0; BitLength_8040 = 32; Address_ = '%QD69'; TYPE_ = 'DINT'; Address_Pointer = ADR(%QD69); AdrOffset_8050 = 292; BitOffset_8050 = 0; BitLength_8050 = 32; Address_ = '%QD73'; TYPE_ = 'UDINT'; Address_Pointer = ADR(%QD73); AdrOffset_8060 = 0; BitOffset_8060 = 0; BitLength_8060 = 0; Address_ = ''; TYPE_ = '';
                  Address_Pointer = 0; AdrOffset_8070 = 0; BitOffset_8070 = 0; BitLength_8070 = 0; Address_ = ''; TYPE_ = ''; Address_Pointer = 0; AdrOffset_8080 = 0; BitOffset_8080 = 0; BitLength_8080 = 0; Address_ = ''; TYPE_ = ''; Address_Pointer = 0; AdrOffset_8510 = 272; BitOffset_8510 = 0; BitLength_8510 = 16; Address_ = '%IW136'; TYPE_ = 'UINT'; Address_Pointer = ADR(%IW136); AdrOffset_8520 = 280; BitOffset_8520 = 0; BitLength_8520 = 32; Address_ = '%ID70'; TYPE_ = 'DINT'; Address_Pointer = ADR(%ID70); AdrOffset_8530 = 278; BitOffset_8530 = 0; BitLength_8530 = 8; Address_ = '%IB278'; TYPE_ = 'SINT'; Address_Pointer = ADR(%IB278); AdrOffset_8540 = 0; BitOffset_8540 = 0; BitLength_8540 = 0; Address_ = ''; TYPE_ = ''; Address_Pointer = 0; AdrOffset_8550 = 0; BitOffset_8550 = 0; BitLength_8550 = 32;
                  Address_ = 'ActVel_RL'; TYPE_ = 'DINT'; Address_Pointer = ADR(ActVel_RL); AdrOffset_8560 = 0; BitOffset_8560 = 0; BitLength_8560 = 0; Address_ = ''; TYPE_ = ''; Address_Pointer = 0; AdrOffset_8570 = 0; BitOffset_8570 = 0; BitLength_8570 = 0; Address_ = ''; TYPE_ = ''; Address_Pointer = 0
      CAN_Port_1 : CAN Port, Inovance, version 00.00.00.10
          settings: IsFreeCAN = True; DeviceGuid = '41b44ff1-ebbe-4db4-bb20-eb005c34d964'; DeviceName = 'GL20_2CAN'; Port = 32; Type = 41090
        CAN自由协议 : CAN自由协议, Inovance, version 00.00.00.10
            settings: CANBusGeneralStruct.BusNodeID = 32; IsPortSub = True; IsLocalCAN = True; IsFreeCAN = True; DeviceTaskName = 'MainTask'; IsVirtual = True; VirtualInterface = 0; TotalChannelCount = 5; channel0.SendingMethod = False; channel0.FrameType = False; channel0.FrameFormat = False; channel0.FrameID = 361; channel0.NumberOfBytes = 8; channel0.RetransmissionInterval = 20; channel0.CycleSendingTime = 20; channel0.IOMappingParamId = 4285874176; channel1.uiChannelIndex = 1; channel1.SendingMethod = False; channel1.FrameType = False; channel1.FrameFormat = False; channel1.FrameID = 617; channel1.NumberOfBytes = 8; channel1.RetransmissionInterval = 20; channel1.CycleSendingTime = 20; channel1.IOMappingParamId = 4285874177; channel2.uiChannelIndex = 2; channel2.SendingMethod = False; channel2.FrameType = False; channel2.FrameFormat = False; channel2.FrameID = 1977; channel2.NumberOfBytes = 8; channel2.RetransmissionInterval = 5; channel2.CycleSendingTime = 10; channel2.IOMappingParamId = 4285874178; channel3.uiChannelIndex = 3; channel3.SendingMethod = False; channel3.FrameType = False; channel3.FrameFormat = False; channel3.FrameID = 256; channel3.NumberOfBytes = 8;
              channel3.RetransmissionInterval = 5; channel3.CycleSendingTime = 10; channel3.IOMappingParamId = 4285874179; channel4.uiChannelIndex = 4; channel4.SendingMethod = False; channel4.FrameType = False; channel4.FrameFormat = False; channel4.FrameID = 81; channel4.NumberOfBytes = 8; channel4.RetransmissionInterval = 5; channel4.CycleSendingTime = 10; channel4.IOMappingParamId = 4285874180
            input  Application.ReciveCanID : DWORD  // Receive Data.FrameID
            input  Application.ReciveCanData  // Receive Data.FrameFirstAddressArray
            output Application.CAN_SES_Req_Data_F : ARRAY [0..7] OF BYTE  // Channel0
            output Application.CAN_SES_Req_Data_R : ARRAY [0..7] OF BYTE  // Channel1
            output Application.VCU_SEB_Req_Data : ARRAY [0..7] OF BYTE  // Channel2
            output Application.main.fbMoveFSD.BMS_Send_Data : ARRAY [0..7] OF BYTE  // Channel3
            output Application.main.fbMoveFSD.CCU_CAN_Data : ARRAY [0..7] OF BYTE  // Channel4
            unmapped channels: Receive Data
      CAN_Port_2 : CAN Port, Inovance, version 00.00.00.10
          settings: IsFreeCAN = False; DeviceGuid = '41b44ff1-ebbe-4db4-bb20-eb005c34d964'; DeviceName = 'GL20_2CAN'; InterfaceNo = 1; Port = 33; Type = 41090
    Serial : 串行接口, 汇川技术股份有限公司, version 00.00.00.10
      COM : Serial Port, Inovance, version 00.00.00.10
          settings: Device = AM521-0808TP/TN; devGuid = 'e348f94f-2bae-4e83-9430-22bd03696b88'
      COM_1 : Serial Port, Inovance, version 00.00.00.10
          settings: COM = 4; Device = GE20_CAN_485; Type = 1; devGuid = '83de0e76-e450-4053-a235-86c09473ce3d'
    LocalHSIO : 本地高速IO, 汇川技术股份有限公司, version 2.0.0.0
        input  Application.main.fbMoveFSD.IsCollision : BOOL  // DigitalInput.Bit0
        unmapped channels: DigitalInput, DigitalOutput
    EXP_A : 扩展卡, 汇川技术股份有限公司, version 00.00.00.10
      GE20_CAN_485 : GE20_CAN_485, Inovance, version 1.0.0.0
          settings: GE20_CAN_485 ExtCard configure.SerialAlias = 4; GE20_CAN_485 ExtCard configure.CANAlias = 4
    EXP_B : 扩展卡, 汇川技术股份有限公司, version 00.00.00.10
    HwConfiguratioinDevice : SystemConfig, Inovance, version 00.00.00.10
        settings: NetworkConfigArray.NetworkConfigArray.BusType = 10; NetworkConfigArray.NetworkConfigArray.RackSum = 1; NetworkConfigArray.NetworkConfigArray.HardwareConfigArray.HardwareConfigArray.RackNo = 1; NetworkConfigArray.NetworkConfigArray.HardwareConfigArray.HardwareConfigArray.ModuleNum = 1; EnableFun = 1
*)

// Device/Application/GVL
VAR_GLOBAL
	//遥控器参数接收
	YkqTxPDO0_data	:	ARRAY[0..7] OF BYTE;
	YkqTxPDO1_data	:	ARRAY[0..7] OF BYTE;
	YkqRxPDO0_data	:	ARRAY[0..7] OF BYTE;
	DriveBySelf		:	BOOL ;
	DriveByYaokong	:	BOOL ;
	Emergency_Stop	:	BOOL;
	Remote_Break	:	BOOL;
	
	//UDP接收超时触发器
	rtrig_recv: R_TRIG;  // 上升沿触发器
	
	bEStopLatched: BOOL := FALSE;  // 闩锁标志：E-stop后保持停止
    ftrig_EStop: F_TRIG;  // 检测E-stop下降沿（释放）
    rtrig_NewCmd_FSD: R_TRIG;  // FSD模式新命令（UDP接收）
	
	//本体层
	TargetVehicleSpeed	:	LREAL:=5;  //km/h
	TargetVehicleAngle	:	LREAL;
	ActVehicleSpeed		:	LREAL;
	ActVehicleAngle		:	LREAL;
	//电机层
	MaxMotorSpeed	:	UDINT:=1400; //rpm
	(* 反馈 / PDO 映射变量（需绑定 CANopen PDO） *)
    ActPos_FL   : DINT; (* map <- PDO: 前左实际位置 (PDO units) *)
    ActPos_FR   : DINT; (* map <- PDO: 前右实际位置 *)
    ActVel_RL   : DINT; (* map <- PDO: 左后实际角速 (rpm) *)
    ActVel_RR   : DINT; (* map <- PDO: 右后实际角速 (rpm) *)
    (* 最终下发变量（绑定到 PDO -> 驱动），类型为 DINT 与驱动匹配 *)
    PDO_TargetPos_FL : DINT; (* map -> PDO *)
    PDO_TargetPos_FR : DINT;
    PDO_TargetVel_RL : DINT; (* rpm *)
    PDO_TargetVel_RR : DINT; (* rpm *)
	
	// 转向系统
     CAN_SES_Req_R : FB_CAN_VCU_SES_Req;
     CAN_SES_Req_F : FB_CAN_VCU_SES_Req;
	 CAN_SES_Req_Data_F : ARRAY[0..7] OF BYTE;
     CAN_SES_Req_Data_R : ARRAY[0..7] OF BYTE;
	 //制动系统
	 VCU_SEB_Req_Data : ARRAY[0..7] OF BYTE;
	
	//单、双阿克曼切换标志
	//True 是单阿克曼、FALSE是双阿克曼
	AckermanModleTransfer	:	BOOL;
	
	ReciveCanData	:	ARRAY[0..7] OF BYTE;
	ReciveCanID		:	DWORD;
END_VAR

// Device/Application/main
PROGRAM main
VAR
    (* 上层命令 *)
    v_cmd_top      : LREAL := 0.0;   // m/s
    delta_cmd_top  : LREAL := 0.0;   // rad

    (* FB 实例 *)
	test		: test;
    fbKine      : FB_AckermannKinematics;
    fbLimiter   : FB_CommandLimiter;
    fbSteer     : FB_SteerPositionPID;
    fbRearPID   : FB_RearWheelVelocityPID;
	fbInvKine	: FB_AckermannInverseKinematics;
	fbUdp		: FB_UDP;
	fbTest		: FB_Test;

	fbMoveYkq	: FB_MoveByYaokong;
	fbMoveFSD	: FB_MoveByFSD;
	recvBuf     : ARRAY[0..12] OF BYTE;
	sendBuf     : ARRAY[0..12] OF BYTE := [0,0,0,0,0,0,0,0,0,0,0,0];
	
	cantest	:	cantesttest;
	udpTimeOut	:	BOOL:=FALSE;
	
END_VAR

(* 1) 运动学计算 *)
v_cmd_top := TargetVehicleSpeed;
delta_cmd_top := TargetVehicleAngle;
fbKine(v_kmh := v_cmd_top, delta := delta_cmd_top);

(* 2) 限幅 最大转角27°*)  
fbLimiter(
    deltaL_in := fbKine.deltaL,
    deltaR_in := fbKine.deltaR,
    omegaRL_in := fbKine.wRL_rpm,
    omegaRR_in := fbKine.wRR_rpm,
    delta_max := 0.47123889,  
    vel_max_rad := 4000
);

(* 3) 前轮转角 PID（位置模式） *)
fbSteer(
    deltaL_ref := fbLimiter.deltaL_lim,
    deltaR_ref := fbLimiter.deltaR_lim,
    dt_ := 0.01,
    Kp := 8.0,
    Ki := 1.0,
    Kd := 0.1,
    outMax := 1000.0,
    outMin := -1000.0,
    derivTau := 0.02,
    usePositionSetpoint := TRUE,
    PosUnitPerRad := 180.0/3.14159265358979323846, // deg/rad or counts_per_rad
    VelUnitPerRadSecToPDO := 60.0/(2.0*3.14159265358979323846),
    ActPos_FL := ActPos_FL,  // VAR_IN_OUT 绑定 (DINT)
    ActPos_FR := ActPos_FR
);

(* 把前轮目标位置写到 PDO 变量 (DINT) *)
PDO_TargetPos_FL := fbSteer.PDO_TargetPos_FL;
PDO_TargetPos_FR := fbSteer.PDO_TargetPos_FR;

(* 4) 后轮速度 PID *)
fbRearPID(
    omegaRL_ref := fbLimiter.omegaRL_lim,
    omegaRR_ref := fbLimiter.omegaRR_lim,
    dt_ := 0.01,
    Kp := 2.5,
    Ki := 0,
    Kd := 0,
    outMax := 3000.0,
    outMin := -3000.0,
    derivTau := 0.02,
    ActVel_RL := ActVel_RL,  // VAR_IN_OUT 绑定 (DINT)
    ActVel_RR := ActVel_RR
);

(* 下发后轮目标速度到 PDO (DINT, rpm) *)
PDO_TargetVel_RL := fbRearPID.PDO_TargetVel_RL;
PDO_TargetVel_RR := fbRearPID.PDO_TargetVel_RR;


fbInvKine(
	ActVel_RL:=ActVel_RL,
	ActVel_RR:=ActVel_RR,
	SteerAngle_FL:=PDO_TargetPos_FL,
	SteerAngle_FR:=PDO_TargetPos_FR
);
//ActVehicleAngle := fbInvKine.HeadingAngle;
ActVehicleSpeed := fbInvKine.VehicleSpeed;


//////////////////////////////////////////////////////////////////////////////////////////
// E-stop闩锁统一处理（放在主循环开头）
ftrig_EStop(CLK := GVL.Emergency_Stop);  // 检测释放（下降沿）

IF GVL.Emergency_Stop THEN
    GVL.bEStopLatched := TRUE;  // 激活闩锁
ELSIF ftrig_EStop.Q THEN
    // 释放时，确保闩锁已设（冗余）
    GVL.bEStopLatched := TRUE;
END_IF

// 根据模式重置闩锁（稍后在FB中检测新命令）

//测试使用

IF DriveBySelf THEN
	cantest();
	fbUdp(sendBuf:=sendBuf, recvBuf=>recvBuf, bNoRecvTimeout=>udpTimeOut);
	fbMoveFSD(udpRxTimeOut:=udpTimeOut, Initial := TRUE ,UDP_RecvBuf := recvBuf, UDP_SendBuf => sendBuf);
	
ELSIF DriveByYaokong THEN
	//遥控器控制
	fbMoveYkq();
	//test();
END_IF

END_PROGRAM

// Device/Application/test
FUNCTION_BLOCK test
VAR_INPUT
END_VAR
VAR_OUTPUT
END_VAR
VAR
	udp : FB_UDP;
	recvBuf     : ARRAY[0..12] OF BYTE;
	sendBuf     : ARRAY[0..12] OF BYTE := [0,1,2,0,0,0,0,0,0,0,0,0];
	
END_VAR



udp(sendBuf := sendBuf, recvBuf=>recvBuf);

END_FUNCTION_BLOCK

// Device/Application/FB_UDP
FUNCTION_BLOCK FB_UDP
VAR_INPUT
	//xEnable     : BOOL;               // 是否使能工作
	sendBuf	 	: ARRAY[0..12] OF BYTE;
END_VAR
VAR_OUTPUT
	recvBuf     : ARRAY[0..12] OF BYTE;
	bNoRecvTimeout: BOOL;
END_VAR
VAR
	UDP_Peer	:	UDP_Peer;
	UDP_Send	:	UDP_Send;
	UDP_Receive	:	UDP_Receive;
	
	IpAddrLocal	:	STRING	:= '192.168.100.210';
	PortLocal	:	UINT	:= 4002;
	hPeer		:	DWORD;
	
	
	remoteIP    : STRING(80) := '192.168.100.10';
	remotePort  : UINT := 8001;
	//sendData	: ARRAY[0..12] OF BYTE := [16#08,SHR(16#51, 24) AND 16#FF,SHR(16#51, 16) AND 16#FF,SHR(16#51, 8) AND 16#FF,SHR(16#51, 0) AND 16#FF,01,00,00,00,00,00,00,00];

	SendErrorID		:	DWORD;
	bSendDone		:	BOOL;
	bSendBusy		:	BOOL;
	bRecvDone		:	BOOL;
	bRecvBusy		:	BOOL;
	
    ton_no_recv: TON;    // 延时接通定时器
    //bNoRecvTimeout: BOOL := FALSE;  // 输出布尔信号：TRUE表示0.5秒内无数据接收
	//recvBuf     : ARRAY[0..15] OF BYTE;
	
	fbPWM	:	FB_PWM;
	pwm	:	BOOL;
	//rTrigSend : R_TRIG;
	PeerErrorID: DWORD;
END_VAR


UDP_Peer(
	xEnable:=TRUE,
	strIpAddrLocal:=IpAddrLocal,
	uiPortLocal:=PortLocal,
	dwErrorID =>PeerErrorID);

	
hPeer := UDP_Peer.hPeer;

	//接收
UDP_Receive(xEnable:=TRUE,
		hPeer := hPeer,
		uiSize := SIZEOF(recvBuf),
		pbyData := ADR(recvBuf),
		xBusy => bRecvDone,
		xDone => bRecvBusy
		);

	//发送
fbPWM(Enable:=TRUE);
pwm := fbPWM.PWM;
	
UDP_Send(xExecute:=pwm,
	hPeer := hPeer,
	strIpAddrDst := remoteIP,
	uiPortDst := remotePort,
	uiSize := SIZEOF(sendBuf),
	pbyData := ADR(sendBuf),
	udiTimeOut:=500000,
	dwErrorID => SendErrorID,
	xDone	=>	bSendDone,
	xBusy	=>	bSendBusy
);	

// 新增逻辑：0.5秒无接收数据检测
rtrig_recv(CLK := bRecvDone);  // 检测接收完成的上升沿

IF rtrig_recv.Q THEN
    ton_no_recv.IN := FALSE;   // 重置定时器
    ton_no_recv(PT := T#500ms);
ELSE
    ton_no_recv.IN := TRUE;    // 正常计时
    ton_no_recv(PT := T#500ms);
END_IF

bNoRecvTimeout := ton_no_recv.Q;  // 输出信号：超时为TRUE

END_FUNCTION_BLOCK

// Device/Application/FB_PWM
FUNCTION_BLOCK FB_PWM
VAR_INPUT
	Enable     : BOOL := TRUE;        // 使能输出
    HalfPeriod : TIME := T#500ms;     // 半周期（默认500ms -> 总周期1s）
END_VAR
VAR_OUTPUT
	PWM        : BOOL := FALSE;       // 输出的PWM布尔量
END_VAR
VAR
	tmr : TON;                        // 定时器（标准TON）
END_VAR

IF NOT Enable THEN
    PWM := FALSE;
    tmr(IN := FALSE);    // 停止并复位定时器
ELSE
    // 定时器启动：计时到达 HalfPeriod 时 tmr.Q = TRUE
    tmr(IN := TRUE, PT := HalfPeriod);

    IF tmr.Q THEN
        // 到达半周期：翻转PWM并复位定时器以开始下一半周期
        PWM := NOT PWM;
        tmr(IN := FALSE);    // 复位定时器（下一循环会再设为 TRUE 重启计时）
    END_IF
END_IF

END_FUNCTION_BLOCK

// Device/Application/FB_AckermannKinematics
FUNCTION_BLOCK FB_AckermannKinematics
VAR_INPUT
	v_kmh		:	LREAL;	//前进速度（km/h)，车辆质心
	delta	:	LREAL;	//等效前轮转角（rad）
	Dir_LR 	: BYTE;
END_VAR
VAR_OUTPUT
	deltaL  : LREAL;  // 左前轮转角 (rad)
    deltaR  : LREAL;  // 右前轮转角 (rad)
    wRL_rpm     : LREAL;  // 左后轮角速度 (rpm)
    wRR_rpm     : LREAL;  // 右后轮角速度 (rpm)
	radius   : LREAL;   // 转弯半径
END_VAR

VAR
	v_ms   :	LREAL;	//前进速度m/s
	L   : LREAL := 1.4;   // 轴距 m
    W   : LREAL := 1.150;   // 轮距 m
    rRL : LREAL := 0.245;   // 左后轮半径 m
    rRR : LREAL := 0.245;   // 右后轮半径 m
    eps : LREAL := 1E-6;   // 防止除零
	
	
    psiDot  : LREAL;   // 偏航角速度 rad/s
    vRL     : LREAL;   // 左后轮线速度
    vRR     : LREAL;   // 右后轮线速度
	tmp 	: LREAL;
	
END_VAR



v_ms := v_kmh / 3.6;  // km/h  ->  m/s

IF ABS(delta) < eps THEN
	radius := 1.0E12;  
	psiDot := 0;
	deltaL := 0;
	deltaR := 0;
	vRL := v_ms;
	vRR := v_ms;
ELSE
	radius := ABS(L / TAN(delta));  //根据自行车模型算出车体转弯半径
	psiDot := v_ms / radius;
	
	deltaL := ATAN(L/2/(radius-W/2)); // 双阿克曼，前后轮转角相同，所以只以前轮计算
	deltaR := ATAN(L/2/(radius+W/2));
	
	vRL := psiDot * SQRT( EXPT((radius - W/2),2) + EXPT(L/2,2) ); //车轮的线速度 m/s
	vRR := psiDot * SQRT( EXPT((radius + W/2),2) + EXPT(L/2,2) );
END_IF

IF Dir_LR  = 2 THEN //右转
	tmp := vRL;
	vRL := vRR;
	vRR := tmp;
END_IF

wRL_rpm := vRL / rRL * 60 / (2*3.1415926);  //车轮转速 rpm
wRR_rpm := vRR / rRR * 60 / (2*3.1415926);

END_FUNCTION_BLOCK

// Device/Application/FB_CommandLimiter
FUNCTION_BLOCK FB_CommandLimiter
VAR_INPUT
	deltaL_in      : LREAL;   // 输入：左前轮目标角（rad）
    deltaR_in      : LREAL;   // 输入：右前轮目标角（rad）
    omegaRL_in     : LREAL;   // 输入：左后轮目标角速（rad/s）
    omegaRR_in     : LREAL;   // 输入：右后轮目标角速（rad/s）
    delta_max      : LREAL := 0.5235987756; // 前轮最大机械角 (rad)
    vel_max_rad    : LREAL := 4000.0;        // 电机最大角速 (rpm)
END_VAR
VAR_OUTPUT
	deltaL_lim     : LREAL;   // 输出：限幅后左前轮角 (rad)
    deltaR_lim     : LREAL;   // 输出：限幅后右前轮角 (rad)
    omegaRL_lim    : LREAL;   // 输出：限幅后左后轮角速 (rad/s)
    omegaRR_lim    : LREAL;   // 输出：限幅后右后轮角速 (rad/s)
END_VAR
VAR
END_VAR

(* 前轮角度限幅 *)
deltaL_lim := deltaL_in;
deltaR_lim := deltaR_in;
IF deltaL_lim > delta_max THEN deltaL_lim := delta_max; END_IF
IF deltaL_lim < -delta_max THEN deltaL_lim := -delta_max; END_IF
IF deltaR_lim > delta_max THEN deltaR_lim := delta_max; END_IF
IF deltaR_lim < -delta_max THEN deltaR_lim := -delta_max; END_IF

(* 后轮角速度限幅 *)
omegaRL_lim := omegaRL_in;
omegaRR_lim := omegaRR_in;
IF omegaRL_lim > vel_max_rad THEN omegaRL_lim := vel_max_rad; END_IF
IF omegaRL_lim < -vel_max_rad THEN omegaRL_lim := -vel_max_rad; END_IF
IF omegaRR_lim > vel_max_rad THEN omegaRR_lim := vel_max_rad; END_IF
IF omegaRR_lim < -vel_max_rad THEN omegaRR_lim := -vel_max_rad; END_IF

END_FUNCTION_BLOCK

// Device/Application/FB_SteerPositionPID
FUNCTION_BLOCK FB_SteerPositionPID
VAR_INPUT
    deltaL_ref    : LREAL;   // 期望左前轮角度 (rad)
    deltaR_ref    : LREAL;   // 期望右前轮角度 (rad)
    dt_           : LREAL := 0.01; // 控制周期 (s)
    Kp            : LREAL := 8.0;
    Ki            : LREAL := 1.0;
    Kd            : LREAL := 0.1;
    outMax        : LREAL := 1000.0;  // 速度模式输出上限 (rpm 等)
    outMin        : LREAL := -1000.0;
    derivTau      : LREAL := 0.02;
    usePositionSetpoint : BOOL := TRUE; // TRUE: 下发位置 setpoint(TRUE：位置模式； FALSE：速度模式)
    PosUnitPerRad : LREAL := 180.0/3.14159265358979323846; // 默认 deg/rad，若你的驱动用 counts 把这里改为 counts_per_rad
    VelUnitPerRadSecToPDO : LREAL := 60.0/(2.0*3.14159265358979323846); // rad/s -> rpm
END_VAR

VAR_IN_OUT
    ActPos_FL     : DINT;   // 
    ActPos_FR     : DINT;   // 
END_VAR

VAR_OUTPUT
    PDO_TargetPos_FL : DINT; //
    PDO_TargetPos_FR : DINT;
    PDO_TargetVel_FL : DINT; // 
    PDO_TargetVel_FR : DINT;
END_VAR

VAR
    actPosRadL   : LREAL;
    actPosRadR   : LREAL;
    errL, errR   : LREAL;
    prevErrL     : LREAL := 0.0;
    prevErrR     : LREAL := 0.0;
    integralL    : LREAL := 0.0;
    integralR    : LREAL := 0.0;
    derivL_filt  : LREAL := 0.0;
    derivR_filt  : LREAL := 0.0;
    alpha        : LREAL;
    deriv_rawL   : LREAL;
    deriv_rawR   : LREAL;
    pidOutL      : LREAL; // 若输出速度则单位为 rad/s (需乘 conversion)
    pidOutR      : LREAL;
    PI_CONST     : LREAL := 3.14159265358979323846;
END_VAR

IF dt_ <= 0.0 THEN dt_ := 0.01; END_IF
alpha := derivTau / (derivTau + dt_);

(* 将 ActPos (DINT, PDO units) 转为弧度 *)
actPosRadL := DINT_TO_LREAL(ActPos_FL) / PosUnitPerRad; 
actPosRadR := DINT_TO_LREAL(ActPos_FR) / PosUnitPerRad; 

(* 位置环 PID（rad 域） *)
errL := deltaL_ref - actPosRadL;
integralL := integralL + errL * dt_;
deriv_rawL := (errL - prevErrL) / dt_;
derivL_filt := alpha * derivL_filt + (1.0 - alpha) * deriv_rawL;
pidOutL := Kp * errL + Ki * integralL + Kd * derivL_filt;

IF pidOutL > outMax THEN
    pidOutL := outMax;
    integralL := integralL - errL * dt_;
ELSIF pidOutL < outMin THEN
    pidOutL := outMin;
    integralL := integralL - errL * dt_;
END_IF
prevErrL := errL;

errR := deltaR_ref - actPosRadR;
integralR := integralR + errR * dt_;
deriv_rawR := (errR - prevErrR) / dt_;
derivR_filt := alpha * derivR_filt + (1.0 - alpha) * deriv_rawR;
pidOutR := Kp * errR + Ki * integralR + Kd * derivR_filt;

IF pidOutR > outMax THEN
    pidOutR := outMax;
    integralR := integralR - errR * dt_;
ELSIF pidOutR < outMin THEN
    pidOutR := outMin;
    integralR := integralR - errR * dt_;
END_IF
prevErrR := errR;

(* 输出 *)
IF usePositionSetpoint THEN
    (* 位置模式：把目标角（rad）转换为 PDO 单位 (PosUnitPerRad)，然后 LREAL->DINT *)
    PDO_TargetPos_FL := LREAL_TO_DINT( deltaL_ref * PosUnitPerRad );  
    PDO_TargetPos_FR := LREAL_TO_DINT( deltaR_ref * PosUnitPerRad );  
    PDO_TargetVel_FL := 0;
    PDO_TargetVel_FR := 0;
ELSE
    (* 速度模式：把 pidOut (rad/s) 转换为 PDO 速度单位 (rpm) *)
    (* 先把 pidOut（rad/s）乘以系数转换为 rpm，再 LREAL->DINT *)
    PDO_TargetVel_FL := LREAL_TO_DINT( pidOutL * VelUnitPerRadSecToPDO ); 
    PDO_TargetVel_FR := LREAL_TO_DINT( pidOutR * VelUnitPerRadSecToPDO ); 
    PDO_TargetPos_FL := 0;
    PDO_TargetPos_FR := 0;
END_IF

END_FUNCTION_BLOCK

// Device/Application/FB_RearWheelVelocityPID
FUNCTION_BLOCK FB_RearWheelVelocityPID
VAR_INPUT
    omegaRL_ref   : LREAL;   // 左后轮目标角速 (rad/s)
    omegaRR_ref   : LREAL;   // 右后轮目标角速 (rad/s)
    dt_           : LREAL := 0.01;
    Kp            : LREAL := 5;
    Ki            : LREAL := 0;
    Kd            : LREAL := 0;
    outMax        : LREAL := 3000.0;  // 最大输出(rpm)，调为合适值
    outMin        : LREAL := -3000.0;
    derivTau      : LREAL := 0.02;
END_VAR

VAR_IN_OUT
    ActVel_RL     : DINT;   // <<< 修改：来自 PDO 反馈 (rpm) (DINT)
    ActVel_RR     : DINT;   // <<< 修改：来自 PDO 反馈 (rpm) (DINT)
END_VAR

VAR_OUTPUT
    PDO_TargetVel_RL : DINT; // <<< 修改：下发给驱动 (rpm) (DINT)
    PDO_TargetVel_RR : DINT; // <<< 修改
END_VAR

VAR
    (* 内部以 LREAL 进行 PID 运算，单位为 rpm *)
    rpmRefRL      : LREAL;
    rpmRefRR      : LREAL;
    actRPM_RL     : LREAL;
    actRPM_RR     : LREAL;
    errRL, errRR  : LREAL;
    prevErrRL     : LREAL := 0.0;
    prevErrRR     : LREAL := 0.0;
    integralRL    : LREAL := 0.0;
    integralRR    : LREAL := 0.0;
    derivFiltRL   : LREAL := 0.0;
    derivFiltRR   : LREAL := 0.0;
    alpha         : LREAL;
    deriv_rawRL   : LREAL;
    deriv_rawRR   : LREAL;
    pidOutRL      : LREAL;
    pidOutRR      : LREAL;
    u_raw_RL      : LREAL;
    u_raw_RR      : LREAL;
    u_cmd_RL      : LREAL;
    u_cmd_RR      : LREAL;
    PI_CONST      : LREAL := 3.14159265358979323846;
    convVel       : LREAL; // 转换系数：rad/s -> rpm = 60/(2*pi)
END_VAR

(* 保护 *)
IF dt_ <= 0.0 THEN dt_ := 0.01; END_IF
alpha := derivTau / (derivTau + dt_);
convVel := 60.0 / (2.0 * PI_CONST); // rad/s -> rpm

(* 1) 参考角速 rad/s -> rpm *)
rpmRefRL := omegaRL_ref * convVel;   // LREAL
rpmRefRR := omegaRR_ref * convVel;

(* 2) 反馈 DINT -> LREAL (rpm) *)
actRPM_RL := DINT_TO_LREAL(ActVel_RL);       // <<< 修改：显式转换 DINT -> LREAL
actRPM_RR := DINT_TO_LREAL(ActVel_RR);       // <<< 修改

(* 左轮 PID（单位：rpm） *)
errRL := rpmRefRL - actRPM_RL;                       // 目标 - 实测 (rpm)
integralRL := integralRL + errRL * dt_;
deriv_rawRL := (errRL - prevErrRL) / dt_;
derivFiltRL := alpha * derivFiltRL + (1.0 - alpha) * deriv_rawRL;
pidOutRL := Kp * errRL + Ki * integralRL + Kd * derivFiltRL;

(* 抗饱和：若 pidOut 超限则回退积分 *)
u_raw_RL := rpmRefRL + pidOutRL;   // 运动学前馈 + PID 修正 (rpm)
IF u_raw_RL > outMax THEN
    u_cmd_RL := outMax;
ELSIF u_raw_RL < outMin THEN
    u_cmd_RL := outMin;
ELSE
    u_cmd_RL := u_raw_RL;
END_IF

(* 选用简单抗积分风up：当饱和且误差驱动方向使积分继续发散时回退积分 *)
IF (u_cmd_RL <> u_raw_RL) THEN
    (* 饱和，做积分回退 *)
    integralRL := integralRL - errRL * dt_;
END_IF

prevErrRL := errRL;

(* 右轮 PID（单位：rpm） *)
errRR := rpmRefRR - actRPM_RR;
integralRR := integralRR + errRR * dt_;
deriv_rawRR := (errRR - prevErrRR) / dt_;
derivFiltRR := alpha * derivFiltRR + (1.0 - alpha) * deriv_rawRR;
pidOutRR := Kp * errRR + Ki * integralRR + Kd * derivFiltRR;

u_raw_RR := rpmRefRR + pidOutRR;
IF u_raw_RR > outMax THEN
    u_cmd_RR := outMax;
ELSIF u_raw_RR < outMin THEN
    u_cmd_RR := outMin;
ELSE
    u_cmd_RR := u_raw_RR;
END_IF

IF (u_cmd_RR <> u_raw_RR) THEN
    integralRR := integralRR - errRR * dt_;
END_IF

prevErrRR := errRR;

(* 3) 输出：转换为 DINT 并下发到 PDO (rpm) *)
(* 注意：DINT(...) 有截断行为，请确保 outMax/outMin 在 DINT 可表示范围内 *)
PDO_TargetVel_RL := LREAL_TO_DINT(u_cmd_RL);  // <<< 修改：显式转换为 DINT
PDO_TargetVel_RR := LREAL_TO_DINT(u_cmd_RR);  // <<< 修改

// IF PDO_TargetVel_RL > GVL.MaxMotorSpeed THEN
// 	PDO_TargetVel_RL := GVL.MaxMotorSpeed;
// END_IF
// 
// IF PDO_TargetVel_RR > GVL.MaxMotorSpeed THEN
// 	PDO_TargetVel_RR := GVL.MaxMotorSpeed;
// END_IF

END_FUNCTION_BLOCK

// Device/Application/FB_AckermannInverseKinematics
FUNCTION_BLOCK FB_AckermannInverseKinematics
VAR_INPUT
	ActVel_RL    : DINT;   // 左后轮速度反馈 rpm
    ActVel_RR    : DINT;   // 右后轮速度反馈 rpm
    SteerAngle_FL: LREAL;  // 左前轮转角 (rad)
    SteerAngle_FR: LREAL;  // 右前轮转角 (rad)
	radius		 : LREAL;   		//转弯半径
END_VAR
VAR_OUTPUT
	VehicleSpeed : REAL; // 车辆质心速度 (km/h)
	delta		: REAL;  //车轮转向角
    //HeadingAngle : LREAL; // 航向角 (rad)
END_VAR
VAR
	L	:	REAL := 1.4;  //轴距
	v_RL, v_RR   : REAL; // 后轮线速度
    v_rear       : LREAL; // 后轴平均速度
    R_L, R_R     : LREAL; // 由左右前轮计算的转弯半径
    R_avg        : LREAL; // 平均转弯半径
	
	wheelRadius  : LREAL:= 0.245;  // 车轮半径 (m)
    axleLength   : LREAL := 1.4;  // 前后轴距 (m)
    trackWidth   : LREAL := 1.150;  // 前轮轮距 (m)
	eps : LREAL := 1E-6;   // 防止除零
	
	cosL    : REAL;
    cosR    : REAL;
	delta_L     : REAL;   // 左前=左后轮转角 [rad]，正值向左转
    delta_R     : REAL;   // 右前=右后轮转角 [rad]，正值向右转
END_VAR

// ============= 逆运动学计算 =============
IF ActVel_RL < 0 THEN
	ActVel_RL := -ActVel_RL;
END_IF
IF ActVel_RR < 0 THEN
	ActVel_RR := -ActVel_RR;
END_IF
// 1. 单位换算：rpm -> m/s
v_RL := DINT_TO_REAL(ActVel_RL) / 60.0 * 2.0 * 3.14159 * wheelRadius;
v_RR := DINT_TO_REAL(ActVel_RR) / 60.0 * 2.0 * 3.14159 * wheelRadius;

delta_L := ATAN((L/2) / (radius-trackWidth/2));
delta_R := ATAN((L/2) / (radius+trackWidth/2));


// 2. 核心公式：纵向速度 = 左右后轮纵向分速平均
cosL := COS(delta_L);
cosR := COS(delta_R);
// 防止 cos 接近0时数值爆炸（极端蟹行）
IF cosL < 0.05 THEN cosL := 0.05; END_IF;
IF cosR < 0.05 THEN cosR := 0.05; END_IF;

VehicleSpeed := (v_RL * cosL + v_RR * cosR) / 2.0 * 3.6;  //km/h

delta := ATAN((L/2)/radius);

END_FUNCTION_BLOCK

// Device/Application/FB_Test
FUNCTION_BLOCK FB_Test
	
VAR_INPUT
	Start	:	BOOL;
	PDO_TargetVel_RL : DINT; (* rpm *)
    PDO_TargetVel_RR : DINT; (* rpm *)
END_VAR
	
VAR_OUTPUT
END_VAR

VAR
	fbPower_1	:	MC_Power_CO;
	fbMoveVel_1	:	MC_MoveVelocity_CO;

	fbPower_2	:	MC_Power_CO;
	fbMoveVel_2	:	MC_MoveVelocity_CO;

	rTrigStart_RR	:	R_TRIG;
	rTrigStart_RL	:	R_TRIG;
	preSpeed_RL	:	DINT:=0;
	preSpeed_RR	:	DINT:=0;
	speedChanged_RR: BOOL;
	speedChanged_RL: BOOL;
END_VAR

fbPower_1(Axis:=Rr_Wheel,Enable:=TRUE,bRegulatorOn:=TRUE,bDriveStart:=TRUE);
fbPower_2(Axis:=Rl_Wheel,Enable:=TRUE,bRegulatorOn:=TRUE,bDriveStart:=TRUE);

speedChanged_RR := (PDO_TargetVel_RR <> preSpeed_RR);  
rTrigStart_RR(CLK := speedChanged_RR);	
fbMoveVel_1(Axis:=Rr_Wheel,
	Execute:=rTrigStart_RR.Q,
	Velocity:=PDO_TargetVel_RR,
	Acceleration:=10,
	Deceleration:=10);

speedChanged_RL := (PDO_TargetVel_RL <> preSpeed_RL);  
rTrigStart_RL(CLK := speedChanged_RL);
fbMoveVel_2(Axis:=Rl_Wheel,
	Execute:=rTrigStart_RL.Q,
	Velocity:=PDO_TargetVel_RL,
	Acceleration:=10,
	Deceleration:=10);
	
preSpeed_RL:=PDO_TargetVel_RL;
preSpeed_RR:=PDO_TargetVel_RR;

END_FUNCTION_BLOCK

// Device/Application/FB_MoveByYaokong
FUNCTION_BLOCK FB_MoveByYaokong
  VAR_INPUT
  END_VAR

  VAR_OUTPUT
  END_VAR

  VAR
      Dir_FR : BYTE;
      Dir_LR : BYTE;

      targetSpeedMax : LREAL;   // 最大速度
      targetSpeed    : LREAL;   // 实际目标速度（按拨杆比例计算）

      DriveCenter   : INT := 16#7F; // 前后拨杆中位 127
      DriveDeadband : INT := 5;     // 中位死区
      DriveOffset   : INT;          // 相对中位偏移
      DriveRatio    : LREAL;        // 速度比例 0.0~1.0

      Rr_Speed : LREAL;
      Rl_Speed : LREAL;

      fbKine    : FB_AckermannKinematics;
      fbInvKine : FB_AckermannInverseKinematics;

      fbPower_1   : MC_Power_CO;
      fbMoveVel_1 : MC_MoveVelocity_CO;
      fbStop_1    : MC_Stop_CO;

      fbPower_2   : MC_Power_CO;
      fbMoveVel_2 : MC_MoveVelocity_CO;
      fbStop_2    : MC_Stop_CO;

      preSpeed_RL : LREAL := 0.0;   // 上一次下发给左后轮的速度
      preSpeed_RR : LREAL := 0.0;   // 上一次下发给右后轮的速度

      speedChanged_RR : BOOL;
      speedChanged_RL : BOOL;

      ExecuteMove_RR : BOOL := FALSE;
      ExecuteMove_RL : BOOL := FALSE;
      PulseHold_RR   : BOOL := FALSE;
      PulseHold_RL   : BOOL := FALSE;

      Break : BOOL := FALSE;

      

      Ls_mm    : REAL := 100.0;   // 转向节转臂长度 (mm)
      Pitch_mm : REAL := 43.692;  // 转向器线角比 (mm/rev)

      RackTravel_mm : REAL;       // 拉杆位移
      PI            : REAL := 3.1415926;

      RemoteRaw   : BYTE;         // 遥控器左右拨杆原始值 0x00~0xFF
      Ratio       : REAL;         // 归一化比例 0.0~1.0
      SteeringDeg : REAL;         // 前轮转向角度（度）
      SteeringRad : REAL;         // 前轮转角（rad）
      SteerAngle_deg : REAL;      // 转向器目标角度（deg）

      

      // 制动系统
      ParkingButton : BOOL := FALSE;
      ParkingState  : BOOL := FALSE;
      rTrigBtn      : R_TRIG;
      PressureValue : BYTE := 0;
      
  END_VAR

(*
====================================================================
 功能描述：
 1. 解析遥控器 CAN 数据
 2. 计算目标车速与转向角
 3. 进行底盘运动学解算
 4. 下发转向 CAN 报文
 5. 控制驱动轮速度
 6. 处理急停 / 驻车逻辑
====================================================================
*)

(*
====================================================================
 1. 遥控器输入解析
====================================================================
*)
targetSpeedMax := BYTE_TO_LREAL(YkqTxPDO1_data[0]) / 10.0;   // 最大目标速度 km/h
Dir_FR         := YkqTxPDO1_data[1];                         // 前后拨杆
RemoteRaw      := YkqTxPDO1_data[2];                         // 左右拨杆


(*
====================================================================
 2. 前后拨杆 -> 速度比例计算
====================================================================
*)
DriveOffset := BYTE_TO_INT(Dir_FR) - DriveCenter;

IF ABS(DriveOffset) <= DriveDeadband THEN
    DriveRatio := 0.0;
ELSE
    DriveRatio :=
        INT_TO_LREAL(ABS(DriveOffset) - DriveDeadband) /
        INT_TO_LREAL(127 - DriveDeadband);
END_IF;

// 限幅保护
IF DriveRatio > 1.0 THEN
    DriveRatio := 1.0;
ELSIF DriveRatio < 0.0 THEN
    DriveRatio := 0.0;
END_IF;

// 最终目标速度
targetSpeed := targetSpeedMax * DriveRatio;


(*
====================================================================
 3. 左右拨杆 -> 转向计算
====================================================================
*)

// 转向方向
IF RemoteRaw < 127 THEN
    Dir_LR := 1;
ELSE
    Dir_LR := 2;
END_IF;

// 遥控器比例映射
Ratio := BYTE_TO_REAL(RemoteRaw) / 255.0;

// 遥控器值映射为车轮转角
SteeringDeg := -20.0 + (Ratio * 40.0);

// 角度转弧度
SteeringRad := SteeringDeg * 3.1415926 / 180.0;


(*
====================================================================
 4. 转向机构解算
====================================================================
*)

// 轮胎转角 -> 齿条位移
RackTravel_mm := Ls_mm * SteeringRad;

// 齿条位移 -> 转向电机角度
SteerAngle_deg := (RackTravel_mm / Pitch_mm) * 360.0;


(*
====================================================================
 5. 转向 CAN 报文下发
====================================================================
*)

// 前桥转向
CAN_SES_Req_F(
    Tgt_StrAngle    := SteerAngle_deg,
    Tgt_StrAngleSpd := 200,
    Veh_Spd         := 50,
    Enable          := 1
);

CAN_SES_Req_Data_F := CAN_SES_Req_F.CanData;


// 后桥转向（反向）
CAN_SES_Req_R(
    Tgt_StrAngle    := -SteerAngle_deg,
    Tgt_StrAngleSpd := 200,
    Veh_Spd         := 50,
    Enable          := 1
);

CAN_SES_Req_Data_R := CAN_SES_Req_R.CanData;


(*
====================================================================
 6. 底盘运动学解算
====================================================================
*)
fbKine(
    v_kmh := targetSpeed,
    delta := SteeringRad,
    Dir_LR := Dir_LR
);

// 电机转速输出
Rr_Speed :=  fbKine.wRR_rpm;
Rl_Speed := -fbKine.wRL_rpm;     // 左右电机对向安装


(*
====================================================================
 7. 行驶方向处理
====================================================================
*)
IF DriveRatio <= 0.0 THEN

    // 停止
    Rr_Speed := 0.0;
    Rl_Speed := 0.0;

ELSIF DriveOffset < 0 THEN

    // 前进
    // 保持当前方向

ELSE

    // 后退
    Rr_Speed := -Rr_Speed;
    Rl_Speed := -Rl_Speed;

END_IF;


(*
====================================================================
 8. 制动控制
====================================================================
*)
VCU_SEB_Req_Data[0] := 6;
VCU_SEB_Req_Data[3] := PressureValue;


(*
====================================================================
 9. 驱动器上电
====================================================================
*)
fbPower_1(
    Axis          := Rr_Wheel,
    Enable        := TRUE,
    bRegulatorOn  := TRUE,
    bDriveStart   := TRUE
);

fbPower_2(
    Axis          := Rl_Wheel,
    Enable        := TRUE,
    bRegulatorOn  := TRUE,
    bDriveStart   := TRUE
);


(*
====================================================================
 10. 急停逻辑
====================================================================
*)
IF GVL.Emergency_Stop THEN

    Rr_Speed := 0.0;
    Rl_Speed := 0.0;

END_IF;


(*
====================================================================
 11. 驻车按钮逻辑
====================================================================
*)
rTrigBtn(CLK := ParkingButton);

// 按键翻转状态
IF rTrigBtn.Q THEN
    ParkingState := NOT ParkingState;
END_IF;

// 驻车压力控制
IF ParkingState THEN
    PressureValue := 60;
ELSE
    PressureValue := 0;
END_IF;


(*
====================================================================
 12. 速度变化检测
====================================================================
*)
speedChanged_RR := ABS(Rr_Speed - preSpeed_RR) > 0.1;
speedChanged_RL := ABS(Rl_Speed - preSpeed_RL) > 0.1;


(*
====================================================================
 13. Execute 单周期脉冲生成
====================================================================
*)

(*
-----------------------------
 右后轮
-----------------------------
*)
IF PulseHold_RR THEN

    ExecuteMove_RR := FALSE;
    PulseHold_RR   := FALSE;

ELSIF speedChanged_RR THEN

    preSpeed_RR    := Rr_Speed;
    ExecuteMove_RR := TRUE;
    PulseHold_RR   := TRUE;

ELSE

    ExecuteMove_RR := FALSE;

END_IF;


(*
-----------------------------
 左后轮
-----------------------------
*)
IF PulseHold_RL THEN

    ExecuteMove_RL := FALSE;
    PulseHold_RL   := FALSE;

ELSIF speedChanged_RL THEN

    preSpeed_RL    := Rl_Speed;
    ExecuteMove_RL := TRUE;
    PulseHold_RL   := TRUE;

ELSE

    ExecuteMove_RL := FALSE;

END_IF;


(*
====================================================================
 14. 下发速度指令
====================================================================
*)
fbMoveVel_1(
    Axis         := Rr_Wheel,
    Execute      := ExecuteMove_RR,
    Velocity     := Rr_Speed,
    Acceleration := 10,
    Deceleration := 10
);

fbMoveVel_2(
    Axis         := Rl_Wheel,
    Execute      := ExecuteMove_RL,
    Velocity     := Rl_Speed,
    Acceleration := 10,
    Deceleration := 10
);


(*
====================================================================
 15. 底盘反解车速
====================================================================
*)
fbInvKine(
    ActVel_RL     := GVL.ActVel_RL / 10,
    ActVel_RR     := GVL.ActVel_RR / 10,
    SteerAngle_FL := fbKine.deltaL,
    SteerAngle_FR := fbKine.deltaR,
    radius        := fbKine.radius
);


(*
====================================================================
 16. 回传遥控器 PDO 数据
====================================================================
*)
YkqRxPDO0_data[0] := 100;

YkqRxPDO0_data[1] :=
    LREAL_TO_BYTE(fbInvKine.VehicleSpeed);

END_FUNCTION_BLOCK

// Device/Application/FB_MoveByFSD
FUNCTION_BLOCK FB_MoveByFSD
VAR_INPUT
	//recvBuf : ARRAY[0..12] OF BYTE;
	UDP_RecvBuf     : ARRAY[0..12] OF BYTE;
	Initial			:	BOOL;
	udpRxTimeOut	:	BOOL;
END_VAR
VAR_OUTPUT
	UDP_SendBuf     : ARRAY[0..12] OF BYTE;
END_VAR
VAR
	
	fbKine			:	FB_AckermannKinematics;
	fbInvKine		:	FB_AckermannInverseKinematics;
	fbPower_1	:	MC_Power_CO;
	fbMoveVel_1	:	MC_MoveVelocity_CO;
	fbStop_1	:	MC_Stop_CO;
	fbPower_2	:	MC_Power_CO;
	fbMoveVel_2	:	MC_MoveVelocity_CO;
	fbStop_2	:	MC_Stop_CO;
	rTrigStart_RR	:	R_TRIG;
	rTrigStart_RL	:	R_TRIG;
	(* 急停释放检测 *)
    xStopState : BOOL;
    rTrigStopRelease : R_TRIG;
    xExecuteMove_RR : BOOL;
	xExecuteMove_RL : BOOL;
	
	CAN_SCU1_Recv	:	FB_CAN_SCU_1;
	CAN_CCU_Send	:	FB_CAN_CCU;
	CAN_BMS_Send	:	FB_CAN_BMS;
	
	
	//从智驾层接收到的信号
	CANBus_DevRxMsg_0: CANBus_DevRxMsg;
	rx_enable	:	BOOL;
	rx_DexId	:	UINT;
	Rx_FilterMsg	:	CANBus_RxFilter_t;
	RxMsg	:	CANBus_FrameMsg_t;
	error_ID	:	CANBus_FBErrorType_Enum;
	
	
	Target_ForwardWheelAngle	:	LREAL;
	Target_ReardWheelAngleMap		:	LREAL;
	Target_ReardWheelAngle		:	LREAL;
	Target_Speed	:	LREAL;
	//Target_SpeedTest	:	LREAL;
	//Target_ReardWheelAngleTest		:	LREAL;
	
	//给智驾发送的CNA数据
	BMS_Send_Data	:	ARRAY[0..7] OF BYTE;
	CCU_CAN_Data	:	ARRAY[0..7] OF BYTE;
	
	//车体相关参数
	Angle_RL	:	LREAL;
	Angle_RR	:	LREAL;
	Angle_FL	:	LREAL;
	Angle_FR	:	LREAL;
	Speed_RR	:	LREAL;
	Speed_RL	:	LREAL;
	preSpeed_RL	:	LREAL:=0;
	preSpeed_RR	:	LREAL:=0;
	speedChanged_RR: BOOL;
	speedChanged_RL: BOOL;
	Vehicle_Speed	:	REAL;
	Steering_Wheel_Angle	:	REAL;
	radius   : LREAL;   // 转弯半径
	
	
	//触边
	IsCollision	: BOOL := FALSE;
	//刹车
	Break	:	BOOL ;
	//档位
	ShiftLevel	:	UINT;
	
	CanId : UDINT;
	
	test : BOOL := TRUE;
	testSpeed_  : LREAL :=5;
	//转向
	Ls_mm    : REAL := 100.0;   // 转向节转臂长度 (mm)
    Pitch_mm : REAL := 43.692;  // 转向器线角比 (mm/rev)

    RackTravel_mm : REAL;       // 拉杆位移
    PI            : REAL := 3.1415926;
	Ratio       : REAL;         // 归一化比例 0.0~1.0
    //SteeringDeg : REAL;         // 前轮转向角度（度）
    SteeringRad : REAL;         // 前轮转角（rad）
    SteerAngle_deg : REAL;      // 转向器目标角度（deg）
	Target_ReardWheelAngleAbs: LREAL;

    Dir_LR : BYTE;
	
END_VAR

(*
====================================================================
 自动驾驶模式主控制逻辑
 功能：
 1. 自动驾驶初始化
 2. CAN 指令解析
 3. 底盘运动学解算
 4. 驱动轮速度控制
 5. 转向执行
 6. 急停 / 防撞 / 制动逻辑
 7. 整车状态回传
====================================================================
*)

(*
====================================================================
 0. CAN数据接收
====================================================================
*)


(*
====================================================================
 1. 自动驾驶模式初始化
====================================================================
*)
IF Initial THEN

    // 清零历史速度
    preSpeed_RL := 0.0;
    preSpeed_RR := 0.0;

    // 清除初始化标志
    Initial := FALSE;

END_IF;


(*
====================================================================
 2. 驱动器上电
====================================================================
*)
fbPower_1(
    Axis          := Rr_Wheel,
    Enable        := TRUE,
    bRegulatorOn  := TRUE,
    bDriveStart   := TRUE
);

fbPower_2(
    Axis          := Rl_Wheel,
    Enable        := TRUE,
    bRegulatorOn  := TRUE,
    bDriveStart   := TRUE
);


(*
====================================================================
 3. 自动驾驶 CAN 指令解析
====================================================================
*)
//IF ReciveCanID = 16#121 THEN

    // 解析 SCU 控制报文
    CAN_SCU1_Recv(
        RawFrame                      := UDP_RecvBuf,
        SCU_Brk_En                    => Break,
        SCU_Target_Speed              => Target_Speed,
        SCU_Steering_Wheel_Angle_F    => Target_ReardWheelAngleMap,
		SCU_ShiftLevel_Req			  => ShiftLevel
    );

//END_IF;
Target_ReardWheelAngle := Target_ReardWheelAngleMap / 4.444;

//测试使用
//Target_ReardWheelAngle := Target_ReardWheelAngleTest;
(*
====================================================================
 4. 底盘运动学正解
 输入：
    Target_Speed             目标车速
    Target_ReardWheelAngle   目标转角
 输出：
    左右轮转速
    左右轮转角
====================================================================
*)
//增加一个转向方向1,2
Target_ReardWheelAngleAbs := ABS(Target_ReardWheelAngle);
IF Target_ReardWheelAngle >=0 THEN
	Dir_LR := 1;
ELSE
	Dir_LR:=2;
END_IF

fbKine(
    v_kmh  := Target_Speed,
    delta  := Target_ReardWheelAngleAbs,
	Dir_LR := Dir_LR,
    deltaL => Angle_RL,
    deltaR => Angle_RR,

    wRL_rpm => Speed_RL,
    wRR_rpm => Speed_RR,

    radius => radius
);


(*
====================================================================
 5. 单 / 双阿克曼模式切换
====================================================================
*)
IF GVL.AckermanModleTransfer THEN

    // 单阿克曼模式
    Angle_FL := 0.0;
    Angle_FR := 0.0;

ELSE

    // 双阿克曼模式
    Angle_FL := Angle_RL;
    Angle_FR := Angle_RR;

END_IF;


(*
====================================================================
 6. 碰撞保护
====================================================================
*)
IF IsCollision THEN

    Speed_RL := 0.0;
    Speed_RR := 0.0;

END_IF;


(*
====================================================================
 7. 制动 / 急停保护
====================================================================
*)
xStopState := Break OR GVL.Emergency_Stop;

IF xStopState THEN

    Speed_RL := 0.0;
    Speed_RR := 0.0;

END_IF;


(*
====================================================================
 8. 急停闩锁逻辑
 说明：
    急停后保持停车状态，
    直到收到新的 UDP 指令才解除闩锁
====================================================================
*)
GVL.rtrig_NewCmd_FSD(
    CLK := rtrig_recv.Q
);

// IF GVL.bEStopLatched THEN
// 
//     Speed_RL := 0.0;
//     Speed_RR := 0.0;
// 
//     // 收到新控制指令后解除锁定
//     IF GVL.rtrig_NewCmd_FSD.Q THEN
//         GVL.bEStopLatched := FALSE;
//     END_IF;
// 
// END_IF;

(*
====================================================================
 接收数据超时保护
====================================================================
*)
// IF udpRxTimeOut THEN
// 	Speed_RL := 0.0;
//     Speed_RR := 0.0;
// END_IF
(*
====================================================================
档位判断
====================================================================
*)
CASE ShiftLevel OF
	0 :
		Speed_RR :=0;
		Speed_RL :=0;
	2:
		Speed_RR :=0;
		Speed_RL :=0;
	1:
		Speed_RR := -Speed_RR;
		Speed_RL := -Speed_RL;
	3:
		Speed_RR := Speed_RR;
		Speed_RL := Speed_RL;
ELSE
	;
END_CASE

(*
====================================================================
判断是否超过电机最大转速
若超过，则限制转角
====================================================================
*)

(*
====================================================================
 9. 右后轮速度控制
====================================================================
*)

// 速度变化检测
//speedChanged_RR := ABS(ABS(Speed_RR) * 10 - ABS(GVL.ActVel_RR)) >= 2;
speedChanged_RR :=
    ABS(Speed_RR - preSpeed_RR) >= 0.1;

// 上升沿触发 Execute
rTrigStart_RR(
    CLK := speedChanged_RR
);

rTrigStopRelease(
    CLK := NOT xStopState
);
xExecuteMove_RR := rTrigStart_RR.Q OR rTrigStopRelease.Q;
// 下发速度
fbMoveVel_1(
    Axis         := Rr_Wheel,
    Execute      := xExecuteMove_RR,
    Velocity     := Speed_RR,
	//Velocity     := 0,
    Acceleration := 500,
    Deceleration := 500
);


(*
====================================================================
 10. 左后轮速度控制
====================================================================
*)

// 速度变化检测
//speedChanged_RL := ABS(ABS(Speed_RL) *10 - ABS(GVL.ActVel_RL)) >= 2;
speedChanged_RL :=
    ABS(Speed_RL - preSpeed_RL) >= 0.1;

// 上升沿触发 Execute
rTrigStart_RL(
    CLK := speedChanged_RL
);
xExecuteMove_RL	:=	rTrigStart_RL.Q OR rTrigStopRelease.Q;
// 左右电机对向安装
fbMoveVel_2(
    Axis         := Rl_Wheel,
    Execute      := xExecuteMove_RL,
    Velocity     := -Speed_RL,
	//Velocity     := 0,
    Acceleration := 500,
    Deceleration := 500
);


(*
====================================================================
 11. 转向执行
====================================================================
*)

// 角度 -> 弧度
SteeringRad :=
    Target_ReardWheelAngle * 3.1415926 / 180.0;


// 轮胎转角 -> 齿条位移
RackTravel_mm :=
    Ls_mm * SteeringRad;


// 齿条位移 -> 转向器角度
SteerAngle_deg :=
    (RackTravel_mm / Pitch_mm) * 360.0;


(*
--------------------------------------------------------------------
 前桥转向 CAN 报文
--------------------------------------------------------------------
*)
CAN_SES_Req_F(
    Tgt_StrAngle    := SteerAngle_deg,
	//Tgt_StrAngle    := 0,
    Tgt_StrAngleSpd := 200,
    Veh_Spd         := 50,
    Enable          := 1,

    CanData => CAN_SES_Req_Data_F
);


(*
--------------------------------------------------------------------
 后桥转向 CAN 报文
--------------------------------------------------------------------
*)
CAN_SES_Req_R(
    Tgt_StrAngle    := -SteerAngle_deg,
	//Tgt_StrAngle    := 0,
    Tgt_StrAngleSpd := 200,
    Veh_Spd         := 50,
    Enable          := 1,

    CanData => CAN_SES_Req_Data_R
);


(*
====================================================================
 12. 更新历史速度
====================================================================
*)
preSpeed_RL := Speed_RL;
preSpeed_RR := Speed_RR;


(*
====================================================================
 13. 底盘运动学反解
====================================================================
*)
fbInvKine(
    ActVel_RL     := GVL.ActVel_RL / 10,
    ActVel_RR     := GVL.ActVel_RR / 10,

    SteerAngle_FL := fbKine.deltaL,
    SteerAngle_FR := fbKine.deltaR,

    radius        := radius,

    VehicleSpeed  => Vehicle_Speed
);


(*
====================================================================
 14. 整车状态 CAN 回传
====================================================================
*)
CAN_CCU_Send(
    CCU_ShiftLevel_Sts        := 3,
    CCU_P_Sts                 := 1,
    CCU_Ignition_Sts          := 1,
    CCU_Drive_Mode_Shift      := 0,

    Steering_Wheel_Direction  := TRUE,

    CCU_Steering_Wheel_Angle  := fbInvKine.delta,
    CCU_Vehicle_Speed         := fbInvKine.VehicleSpeed,

    CCU_Drive_Mode            := 1,

    Remote_Brake              := test,
    Emergency_Brake           := test,
    SCU_Brake_Singal          := test,

    Left_Turn_Light_Sts       := test,
    Right_Turn_Light_Sts      := test,

    Position_Light_Sts        := test,
    LowBeam_Sts               := test,

    TxFrame => CCU_CAN_Data
);


(*
====================================================================
 15. BMS 状态转发
====================================================================
*)
IF ReciveCanID = 16#444 THEN

    CAN_BMS_Send(
		RxData := ReciveCanData,
        TxData => BMS_Send_Data
    );

END_IF;

END_FUNCTION_BLOCK

// Device/Application/FB_CAN_SCU_1
FUNCTION_BLOCK FB_CAN_SCU_1
VAR_INPUT
	RawFrame : ARRAY[0..12] OF BYTE;   // 13字节原始数据
	
END_VAR
VAR_OUTPUT
	SCU_ShiftLevel_Req	:	UINT;; //底盘档位状态
	SCU_Drive_Mode_Req	:	UINT;; //底盘驾驶模式状态
	SCU_Steering_Wheel_Angle_F	:	SINT; //前转向角度控制
	SCU_Steering_Wheel_Angle_R	:	SINT; //后转向角度控制
	SCU_Target_Speed	:	REAL; //速度控制
	SCU_Brk_En	:	BOOL; //刹车信号控制
	GW_Left_Turn_Light_Req	:	UINT; //左转向灯控制
	GW_Right_Turn_Light_Req	:	UINT; //右转向灯控制
	GW_Position_Light_Req	:	UINT; //刹车灯控制
	GW_LowBeam_Req	:	UINT; //近光灯控制
	angular_speed_flag	:	INT; //调节转向速度，只部分车型适用
	SCU_Brake_Force_Flag	:	BOOL; //调节EMB强度，只针对有EMB的车型
	
END_VAR
VAR
	// 把13字节里真正的8字节CAN数据取出来（第6~13字节，即索引5~12）
    Data : ARRAY[0..7] OF BYTE;
    
    // 64位无符号整数，用于位字段提取（Intel = Little-Endian）
    Raw64 : ULINT;
    
    i : INT;
END_VAR


//============================================================
// 1. 提取真实的8字节CAN数据（跳过前5字节的长度+ID）
//============================================================
FOR i := 0 TO 7 DO
    Data[i] := RawFrame[5 + i];
END_FOR;

//============================================================
// 2. Little-Endian 拼成 64bit 整数（最方便做位操作）
//============================================================
Raw64 :=   (SHL(BYTE_TO_ULINT(Data[7]),56))
         OR (SHL(BYTE_TO_ULINT(Data[6]),48))
         OR (SHL(BYTE_TO_ULINT(Data[5]),40))
         OR (SHL(BYTE_TO_ULINT(Data[4]),32))
         OR (SHL(BYTE_TO_ULINT(Data[3]),24))
         OR (SHL(BYTE_TO_ULINT(Data[2]),16))
         OR (SHL(BYTE_TO_ULINT(Data[1]),8))
         OR  BYTE_TO_ULINT(Data[0]);

//============================================================
// 3. 按协议逐个提取信号（全部是 Intel/Little-Endian）
//============================================================

// Startbit 0, Len 2
SCU_ShiftLevel_Req := ULINT_TO_UINT(SHR(Raw64, 0) AND 16#03);

// Startbit 6, Len 2
SCU_Drive_Mode_Req := ULINT_TO_UINT(SHR(Raw64, 6) AND 16#03);

// Startbit 8, Len 8  → Byte1 的高8位
SCU_Steering_Wheel_Angle_F := ULINT_TO_SINT(SHR(Raw64, 8) AND 16#FF);

// Startbit 16, Len 8 → Byte2
SCU_Steering_Wheel_Angle_R := ULINT_TO_SINT(SHR(Raw64,16) AND 16#FF);

// Startbit 24, Len 9  → 跨Byte3[0..7] + Byte4[0]
SCU_Target_Speed := ULINT_TO_REAL(SHR(Raw64,24) AND 16#1FF) * 0.1;

// Startbit 33, Len 1  → Byte4 的 bit1
SCU_Brk_En := (SHR(Raw64,33) AND 16#01) = 16#01;

// Startbit 40, Len 2 → Byte5 bit0~1
GW_Left_Turn_Light_Req  := ULINT_TO_UINT(SHR(Raw64,40) AND 16#03);

// Startbit 42, Len 2 → Byte5 bit2~3
GW_Right_Turn_Light_Req := ULINT_TO_UINT(SHR(Raw64,42) AND 16#03);

// Startbit 46, Len 2 → Byte5 bit6~7
GW_Position_Light_Req   := ULINT_TO_UINT(SHR(Raw64,46) AND 16#03);

// Startbit 48, Len 2 → Byte6 bit0~1
GW_LowBeam_Req          := ULINT_TO_UINT(SHR(Raw64,48) AND 16#03);

// // Startbit 60, Len 1（有符号） → Byte7 bit4
// angular_speed_flag := IF (SHR(Raw64,60) AND 16#01)=1 THEN 1 ELSE 0; // 实际协议里是Signed，但只有0/1
// 
// // Startbit 60, Len 1（无符号） → 同样位置，另一个信号（两个信号重叠bit）
// SCU_Brake_Force_Flag := (SHR(Raw64,60) AND 16#01) = 16#01;

END_FUNCTION_BLOCK

// Device/Application/FB_CAN_CCU
FUNCTION_BLOCK FB_CAN_CCU
VAR_INPUT
	CCU_ShiftLevel_Sts         : UINT;   // 0~3   档位状态
    CCU_P_Sts                  : BOOL;   // 刹车踏板状态
    CCU_Ignition_Sts           : UINT;   // 0~3   点火状态
    CCU_Drive_Mode_Shift       : BOOL;   // 驾驶模式切换按钮
    Steering_Wheel_Direction   : BOOL;   // 前轮转向方向：TRUE=左转，FALSE=右转
    CCU_Steering_Wheel_Angle   : REAL;   // 实际角度 ° → 发送时×10（协议0.1°/LSB，120→12.0°或27°看标定）
    CCU_Vehicle_Speed          : REAL;   // km/h → 发送时×10（0.1km/h 精度）
    CCU_Drive_Mode             : UINT;   // 0~3   当前驾驶模式
    Remote_Brake               : BOOL;   // 遥控器刹车
    Emergency_Brake            : BOOL;   // 紧急制动
    SCU_Brake_Singal           : BOOL;   // 自动驾驶刹车请求
    Left_Turn_Light_Sts        : BOOL;   // 左转灯实际状态
    Right_Turn_Light_Sts       : BOOL;   // 右转灯实际状态
    Position_Light_Sts         : BOOL;   // 刹车灯状态
    LowBeam_Sts                : BOOL;   // 近光灯状态
END_VAR
VAR_OUTPUT
	TxFrame : ARRAY[0..7] OF BYTE;   // 只有数据
END_VAR
VAR
	Raw64      : ULINT := 0;
	Raw64_CAN      : ULINT := 0;
    angle_raw  : UINT;
    speed_raw  : UINT;
	
	i : INT;
    
	nibble : ULINT;
    
END_VAR

//======================================================
// 1. 按 Intel (Little-Endian) 顺序打包所有信号到 64bit
//======================================================
Raw64 := 0;  // 先清零

// bit 0~1: CCU_ShiftLevel_Sts (2 bits)
Raw64 := Raw64 OR SHL(UINT_TO_ULINT(CCU_ShiftLevel_Sts AND 16#03), 0);

// bit 2: CCU_P_Sts
IF CCU_P_Sts THEN
    Raw64 := Raw64 OR SHL(16#1, 2);
END_IF;

// bit 3~4: CCU_Ignition_Sts (2 bits)
Raw64 := Raw64 OR SHL(UINT_TO_ULINT(CCU_Ignition_Sts AND 16#03), 3);

// bit 5: CCU_Drive_Mode_Shift
IF CCU_Drive_Mode_Shift THEN
    Raw64 := Raw64 OR SHL(16#1, 5);
END_IF;

// bit 7: Steering_Wheel_Direction (左1 右0)
IF Steering_Wheel_Direction THEN
    Raw64 := Raw64 OR SHL(16#1, 7);
END_IF;

// bit 8~19: CCU_Steering_Wheel_Angle (12 bits, 0.1°/LSB)
angle_raw := REAL_TO_UINT(CCU_Steering_Wheel_Angle * 10.0);
Raw64 := Raw64 OR SHL(UINT_TO_ULINT(angle_raw AND 16#0FFF), 8);

// bit 20~28: CCU_Vehicle_Speed (9 bits, 0.1 km/h/LSB)
speed_raw := REAL_TO_UINT(CCU_Vehicle_Speed * 10.0);  // 关键：×10
Raw64 := Raw64 OR SHL(UINT_TO_ULINT(speed_raw AND 16#1FF), 20);

// bit 29~31: CCU_Drive_Mode (3 bits)
Raw64 := Raw64 OR SHL(UINT_TO_ULINT(CCU_Drive_Mode AND 16#07), 29);

// bit 32: Remote_Brake
IF Remote_Brake THEN
    Raw64 := Raw64 OR SHL(16#1, 32);
END_IF;

// bit 33: Emergency_Brake
IF Emergency_Brake THEN
    Raw64 := Raw64 OR SHL(16#1, 33);
END_IF;

// bit 34: SCU_Brake_Singal
IF SCU_Brake_Singal THEN
    Raw64 := Raw64 OR SHL(16#1, 34);
END_IF;

// bit 56: Left_Turn_Light_Sts
IF Left_Turn_Light_Sts THEN
    Raw64 := Raw64 OR SHL(16#1, 56);
END_IF;

// bit 57: Right_Turn_Light_Sts
IF Right_Turn_Light_Sts THEN
    Raw64 := Raw64 OR SHL(16#1, 57);
END_IF;

// bit 59: Position_Light_Sts (刹车灯)
IF Position_Light_Sts THEN
    Raw64 := Raw64 OR SHL(16#1, 59);
END_IF;

// bit 60: LowBeam_Sts
IF LowBeam_Sts THEN
    Raw64 := Raw64 OR SHL(16#1, 60);
END_IF;

//======================================================
// 2. 直接拆出 8 字节数据区（Intel 顺序已经是低字节在前）
//======================================================
TxFrame[0]  := ULINT_TO_BYTE(Raw64);           // Data0
TxFrame[1]  := ULINT_TO_BYTE(SHR(Raw64, 8));    // Data1
TxFrame[2]  := ULINT_TO_BYTE(SHR(Raw64, 16));   // Data2
TxFrame[3]  := ULINT_TO_BYTE(SHR(Raw64, 24));   // Data3
TxFrame[4]  := ULINT_TO_BYTE(SHR(Raw64, 32));   // Data4
TxFrame[5] := ULINT_TO_BYTE(SHR(Raw64, 40));   // Data5
TxFrame[6] := ULINT_TO_BYTE(SHR(Raw64, 48));   // Data6
TxFrame[7] := ULINT_TO_BYTE(SHR(Raw64, 56));   // Data7

//======================================================
// 3. 填充前5字节：DLC + CAN ID 0x51 (Standard Frame)
//    常见格式：Big-Endian ID，标准帧通常低字节有效
//======================================================
// TxFrame[0] := 16#08;         // DLC = 8
// 
// TxFrame[1] := 0;             // ID 高字节
// TxFrame[2] := 0;             
// TxFrame[3] := 0;             
// TxFrame[4] := 16#51;          // ID = 0x51，低字节放这里（常见做法）

END_FUNCTION_BLOCK

// Device/Application/FB_CAN_BMS
FUNCTION_BLOCK FB_CAN_BMS
VAR_INPUT
    RxData : ARRAY[0..7] OF BYTE;
END_VAR

VAR_OUTPUT
    TxData : ARRAY[0..7] OF BYTE;   // 仅仅返回CAN数据
END_VAR

VAR
    (* 原始值 *)
    VoltageRaw : UINT;
    CurrentRaw : INT;

    (* 实际值 *)
    VoltageReal : REAL;
    CurrentReal : REAL;

    (* 重新编码后的值 *)
    VoltageSend : UINT;
    CurrentSend : INT;
END_VAR

(* ============================= *)
(* 1. 解析接收到的CAN数据 *)
(* ============================= *)

(* 电压：低字节在前，高字节在后 *)
VoltageRaw := BYTE_TO_UINT(RxData[0]) OR SHL(BYTE_TO_UINT(RxData[1]), 8);

(* 电流：低字节在前，高字节在后 *)
CurrentRaw := BYTE_TO_INT(RxData[2]) OR SHL(BYTE_TO_INT(RxData[3]), 8);


(* ============================= *)
(* 2. 转换为实际物理量 *)
(* ============================= *)

(* 电压：0~4000 -> 0~400V *)
VoltageReal := UINT_TO_REAL(VoltageRaw) * 0.1;

(* 电流：0~1000 -> -500A~500A *)
CurrentReal := INT_TO_REAL(CurrentRaw) - 500.0;


(* ============================= *)
(* 3. 再重新编码 *)
(* ============================= *)


VoltageSend := REAL_TO_UINT(VoltageReal );
CurrentSend := REAL_TO_INT(CurrentReal );


(* ============================= *)
(* 4. 打包成CAN发送数据 *)
(* ============================= *)

(* 电压 *)
TxData[0] := UINT_TO_BYTE(VoltageSend AND 16#00FF);
TxData[1] := UINT_TO_BYTE(SHR(VoltageSend, 8));

(* 电流 *)
TxData[2] := INT_TO_BYTE(CurrentSend AND 16#00FF);
TxData[3] := INT_TO_BYTE(SHR(CurrentSend, 8));

(* 其余字节清零 *)
TxData[4] := RxData[6];
TxData[5] := 0;
TxData[6] := 0;
TxData[7] := 0;

END_FUNCTION_BLOCK

// Device/Application/cantesttest
FUNCTION_BLOCK cantesttest
VAR_INPUT
END_VAR
VAR_OUTPUT
END_VAR
VAR
	CANBus_CtrlDevState_0: CANBus_CtrlDevState;
	cmd: CANBus_CtrlCmdType_Enum;
	exc: BOOL;
	CANBus_DevRxMsg_0: CANBus_DevRxMsg;
	rxfilter: CANBus_RxFilter_t;
	RxMsg: CANBus_FrameMsg_t;
END_VAR

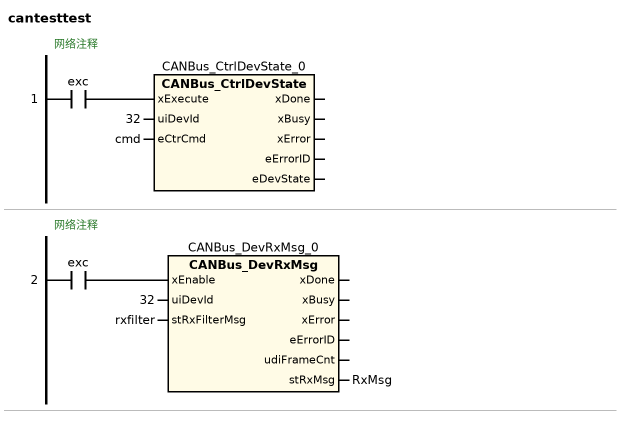
// NETWORK 1
// 网络注释
CANBus_CtrlDevState_0(xExecute := exc, uiDevId := 32, eCtrCmd := cmd); // CANBus_CtrlDevState

// NETWORK 2
// 网络注释
CANBus_DevRxMsg_0(xEnable := exc, uiDevId := 32, stRxFilterMsg := rxfilter, stRxMsg => RxMsg); // CANBus_DevRxMsg

END_FUNCTION_BLOCK

// Device/Application/CANOpen_Task
PROGRAM CANOpen_Task
VAR
END_VAR

END_PROGRAM

// Device/Application/FB_UDP_Recv
FUNCTION_BLOCK FB_UDP_Recv
VAR_INPUT
END_VAR
VAR_OUTPUT
	recvBuf     : ARRAY[0..12] OF BYTE;
END_VAR
VAR
	UDP_Peer	:	UDP_Peer;
	UDP_Send	:	UDP_Send;
	UDP_Receive	:	UDP_Receive;
	
	IpAddrLocal	:	STRING	:= '192.168.100.110';
	PortLocal	:	UINT	:= 4002;
	hPeer		:	DWORD;
	remoteIP    : STRING := '192.168.100.10';
	remotePort  : UINT := 8002;
END_VAR

UDP_Peer(xEnable:=TRUE,
	strIpAddrLocal:=IpAddrLocal,
	uiPortLocal:=PortLocal
	);
	
hPeer := UDP_Peer.hPeer;

//接收
UDP_Receive(xEnable:=TRUE,
		hPeer := hPeer,
		uiSize := SIZEOF(recvBuf),
		pbyData := ADR(recvBuf)
		);

END_FUNCTION_BLOCK

// Device/Application/FB_UDP_Send
FUNCTION_BLOCK FB_UDP_Send
VAR_INPUT
	sendData	 	: ARRAY[0..12] OF BYTE;
END_VAR
VAR_OUTPUT
END_VAR
VAR
	UDP_Peer	:	UDP_Peer;
	UDP_Send	:	UDP_Send;
	UDP_Receive	:	UDP_Receive;
	
	IpAddrLocal	:	STRING	:= '192.168.100.110';
	PortLocal	:	UINT	:= 4002;
	hPeer		:	DWORD;
	remoteIP    : STRING := '192.168.100.10';
	remotePort  : UINT := 8002;
	
	fbPWM	:	FB_PWM;
	pwm	:	BOOL;
	
	ErrorID	:	DWORD;
	bDone	:	BOOL:=FALSE;
	bBu	:	BOOL;
END_VAR


UDP_Peer(xEnable:=TRUE,
			strIpAddrLocal:=IpAddrLocal,
			uiPortLocal:=PortLocal);

hPeer := UDP_Peer.hPeer;
	
fbPWM(Enable:=TRUE);
	pwm := fbPWM.PWM;
	//rTrigSend(CLK := pwm);
	UDP_Send(xExecute:=pwm,
		hPeer := hPeer,
		strIpAddrDst := remoteIP,
		uiPortDst := remotePort,
		uiSize := SIZEOF(sendData),
		pbyData := ADR(sendData),
		udiTimeOut:=500000,
		dwErrorID => ErrorID,
		xDone	=>	bDone,
		xBusy	=>	bBu
		);

END_FUNCTION_BLOCK

// Device/Application/FB_CAN_VCU_SES_Req
FUNCTION_BLOCK FB_CAN_VCU_SES_Req
VAR_INPUT
    Tgt_StrAngle      : REAL;   // 目标转向角（°）
    Tgt_StrAngleSpd   : REAL;   // 目标转向角速度（°/s）
    Veh_Spd           : BYTE;   // 车速（可选，直接填 Byte6）
    Enable            : BOOL;   // 角度控制使能
END_VAR

VAR_OUTPUT
    CanData : ARRAY[0..7] OF BYTE; // 最终 8 字节 CAN 数据
END_VAR

VAR
    RawAngle   : UINT;   // 16bit 原始角度
    RawSpd     : UINT;   // 16bit 原始角速度
    RollCnt    : BYTE;   // 4bit Rolling Counter
    Sum        : UINT;
    i          : INT;
END_VAR

//============================================================
// 1. 物理量 → 原始值
//============================================================

// 角度：Phys = Raw*0.1 - 3000
RawAngle := REAL_TO_UINT((Tgt_StrAngle + 3000.0) / 0.1);

// 角速度：1 °/s per bit
RawSpd := REAL_TO_UINT(Tgt_StrAngleSpd);

//============================================================
// 2. 清空数据
//============================================================
FOR i := 0 TO 7 DO
    CanData[i] := 0;
END_FOR;

//============================================================
// 3. Byte0：控制位
// bit1 = AngleControl_Enable
// bit0 = Alignment_Enable（这里不用，置0）
//============================================================
IF Enable THEN
    CanData[0] := 2;   // 0000 0010
ELSE
    CanData[0] := 0;
END_IF;

//============================================================
// 4. 转向角（Motorola）
// 高字节 → Byte1
// 低字节 → Byte2
//============================================================
CanData[1] := UINT_TO_BYTE(SHR(RawAngle, 8));
CanData[2] := UINT_TO_BYTE(RawAngle AND 16#FF);

//============================================================
// 5. 转向角速度（Motorola）
// 高字节 → Byte3
// 低字节 → Byte4
//============================================================
CanData[3] := UINT_TO_BYTE(SHR(RawSpd, 8));
CanData[4] := UINT_TO_BYTE(RawSpd AND 16#FF);

//============================================================
// 6. Byte5：Rolling Counter + Enable
// bit0 = RollCnt_Enable
// bit1 = CheckSum_Enable
// bit4~7 = Rolling Counter
//============================================================
CanData[5] := 16#03 OR SHL(RollCnt AND 16#0F, 4);

//============================================================
// 7. Byte6：车速
//============================================================
CanData[6] := Veh_Spd;

//============================================================
// 8. Checksum
// CheckSum = (Byte0 + ... + Byte6) XOR 0xFF
//============================================================
Sum := 0;
FOR i := 0 TO 6 DO
    Sum := Sum + CanData[i];
END_FOR;

CanData[7] := UINT_TO_BYTE((Sum AND 16#FF) XOR 16#FF);

//============================================================
// 9. Rolling Counter 自增
//============================================================
RollCnt := (RollCnt + 1) AND 16#0F;

END_FUNCTION_BLOCK
